LIN {X 0,Y 314.134,Z 385.842,A -85,B 0,C 180,E1 15646.01,E2 15646.01} C_VEL
LIN {X 0,Y 314.107,Z 385.802,A -85,B 0,C 180,E1 15641.542,E2 15641.542} C_VEL
LIN {X 0,Y 314.101,Z 385.806,A -85,B 0,C 180,E1 15637.158,E2 15637.158} C_VEL
LIN {X 0,Y 314.157,Z 386.054,A -85,B 0,C 180,E1 15633.754,E2 15633.754} C_VEL
LIN {X 0,Y 314.307,Z 386.869,A -85,B 0,C 180,E1 15633.361,E2 15633.361} C_VEL
LIN {X 0,Y 316.062,Z 390.166,A -85,B 0,C 180,E1 15632.503,E2 15632.503} C_VEL
LIN {X 0,Y 319.649,Z 392.888,A -85,B 0,C 180,E1 15631.061,E2 15631.061} C_VEL
LIN {X 0,Y 322.025,Z 396.633,A -85,B 0,C 180,E1 15629.967,E2 15629.967} C_VEL
LIN {X 0,Y 324.957,Z 398.845,A -85,B 0,C 180,E1 15628.68,E2 15628.68} C_VEL
LIN {X 0,Y 325.868,Z 399.667,A -85,B 0,C 180,E1 15628.262,E2 15628.262} C_VEL
LIN {X 0,Y 328.379,Z 403.252,A -85,B 0,C 180,E1 15626.985,E2 15626.985} C_VEL
LIN {X 0,Y 331.763,Z 405.775,A -85,B 0,C 180,E1 15625.29,E2 15625.29} C_VEL
LIN {X 0,Y 332.732,Z 406.589,A -85,B 0,C 180,E1 15624.775,E2 15624.775} C_VEL
LIN {X 0,Y 335.377,Z 410.277,A -85,B 0,C 180,E1 15623.197,E2 15623.197} C_VEL
LIN {X 0,Y 338.842,Z 412.794,A -85,B 0,C 180,E1 15621.168,E2 15621.168} C_VEL
LIN {X 0,Y 342.057,Z 417.138,A -85,B 0,C 180,E1 15619.111,E2 15619.111} C_VEL
LIN {X 0,Y 345.607,Z 419.696,A -85,B 0,C 180,E1 15616.954,E2 15616.954} C_VEL
LIN {X 0,Y 349.278,Z 424.393,A -85,B 0,C 180,E1 15614.534,E2 15614.534} C_VEL
LIN {X 0,Y 352.998,Z 427.12,A -85,B 0,C 180,E1 15612.104,E2 15612.104} C_VEL
LIN {X 0,Y 355.556,Z 430.698,A -85,B 0,C 180,E1 15610.256,E2 15610.256} C_VEL
LIN {X 0,Y 358.853,Z 433.234,A -85,B 0,C 180,E1 15607.97,E2 15607.97} C_VEL
LIN {X 0,Y 360.061,Z 434.113,A -85,B 0,C 180,E1 15607.103,E2 15607.103} C_VEL
LIN {X 0,Y 362.743,Z 437.733,A -85,B 0,C 180,E1 15604.981,E2 15604.981} C_VEL
LIN {X 0,Y 365.748,Z 440.111,A -85,B 0,C 180,E1 15602.668,E2 15602.668} C_VEL
LIN {X 0,Y 367.537,Z 441.34,A -85,B 0,C 180,E1 15601.213,E2 15601.213} C_VEL
LIN {X 0,Y 369.942,Z 444.728,A -85,B 0,C 180,E1 15599.021,E2 15599.021} C_VEL
LIN {X 0,Y 372.763,Z 447.045,A -85,B 0,C 180,E1 15596.401,E2 15596.401} C_VEL
LIN {X 0,Y 375.125,Z 448.378,A -85,B 0,C 180,E1 15594.15,E2 15594.15} C_VEL
LIN {X 0,Y 377.09,Z 451.528,A -85,B 0,C 180,E1 15591.79,E2 15591.79} C_VEL
LIN {X 0,Y 379.57,Z 453.798,A -85,B 0,C 180,E1 15588.745,E2 15588.745} C_VEL
LIN {X 0,Y 381.929,Z 454.969,A -85,B 0,C 180,E1 15585.487,E2 15585.487} C_VEL
LIN {X 0,Y 383.246,Z 456.112,A -85,B 0,C 180,E1 15583.272,E2 15583.272} C_VEL
LIN {X 0,Y 384.548,Z 458.408,A -85,B 0,C 180,E1 15580.335,E2 15580.335} C_VEL
LIN {X 0,Y 385.649,Z 459.744,A -85,B 0,C 180,E1 15577.149,E2 15577.149} C_VEL
LIN {X 0,Y 386.449,Z 460.442,A -85,B 0,C 180,E1 15573.709,E2 15573.709} C_VEL
LIN {X 0,Y 386.727,Z 460.669,A -85,B 0,C 180,E1 15570.444,E2 15570.444} C_VEL
LIN {X 0,Y 386.569,Z 460.508,A -85,B 0,C 180,E1 15567.035,E2 15567.035} C_VEL
LIN {X 0,Y 385.909,Z 459.957,A -85,B 0,C 180,E1 15563.604,E2 15563.604} C_VEL
LIN {X 0,Y 384.821,Z 458.695,A -85,B 0,C 180,E1 15560.277,E2 15560.277} C_VEL
LIN {X 0,Y 383.571,Z 456.693,A -85,B 0,C 180,E1 15557.352,E2 15557.352} C_VEL
LIN {X 0,Y 382.353,Z 455.172,A -85,B 0,C 180,E1 15555.152,E2 15555.152} C_VEL
LIN {X 0,Y 380.089,Z 454.101,A -85,B 0,C 180,E1 15551.917,E2 15551.917} C_VEL
LIN {X 0,Y 377.688,Z 452.178,A -85,B 0,C 180,E1 15548.898,E2 15548.898} C_VEL
LIN {X 0,Y 375.609,Z 449.353,A -85,B 0,C 180,E1 15546.467,E2 15546.467} C_VEL
LIN {X 0,Y 374.66,Z 447.969,A -85,B 0,C 180,E1 15545.398,E2 15545.398} C_VEL
LIN {X 0,Y 371.406,Z 446.102,A -85,B 0,C 180,E1 15542.315,E2 15542.315} C_VEL
LIN {X 0,Y 368.613,Z 443.116,A -85,B 0,C 180,E1 15539.791,E2 15539.791} C_VEL
LIN {X 0,Y 367.145,Z 440.822,A -85,B 0,C 180,E1 15538.454,E2 15538.454} C_VEL
LIN {X 0,Y 363.643,Z 438.62,A -85,B 0,C 180,E1 15535.692,E2 15535.692} C_VEL
LIN {X 0,Y 360.504,Z 434.893,A -85,B 0,C 180,E1 15533.26,E2 15533.26} C_VEL
LIN {X 0,Y 359.525,Z 433.574,A -85,B 0,C 180,E1 15532.48,E2 15532.48} C_VEL
LIN {X 0,Y 355.99,Z 431.139,A -85,B 0,C 180,E1 15530.048,E2 15530.048} C_VEL
LIN {X 0,Y 353.199,Z 427.491,A -85,B 0,C 180,E1 15528.048,E2 15528.048} C_VEL
LIN {X 0,Y 352.452,Z 426.566,A -85,B 0,C 180,E1 15527.511,E2 15527.511} C_VEL
LIN {X 0,Y 349.115,Z 424.229,A -85,B 0,C 180,E1 15525.359,E2 15525.359} C_VEL
LIN {X 0,Y 346.031,Z 420.14,A -85,B 0,C 180,E1 15523.309,E2 15523.309} C_VEL
LIN {X 0,Y 341.774,Z 416.854,A -85,B 0,C 180,E1 15520.708,E2 15520.708} C_VEL
LIN {X 0,Y 339.259,Z 413.179,A -85,B 0,C 180,E1 15519.089,E2 15519.089} C_VEL
LIN {X 0,Y 335.231,Z 410.123,A -85,B 0,C 180,E1 15516.715,E2 15516.715} C_VEL
LIN {X 0,Y 332.601,Z 406.366,A -85,B 0,C 180,E1 15515.149,E2 15515.149} C_VEL
LIN {X 0,Y 328.555,Z 403.427,A -85,B 0,C 180,E1 15513.099,E2 15513.099} C_VEL
LIN {X 0,Y 325.951,Z 399.829,A -85,B 0,C 180,E1 15511.781,E2 15511.781} C_VEL
LIN {X 0,Y 325.335,Z 399.029,A -85,B 0,C 180,E1 15511.486,E2 15511.486} C_VEL
LIN {X 0,Y 322.117,Z 396.737,A -85,B 0,C 180,E1 15510.075,E2 15510.075} C_VEL
LIN {X 0,Y 319.735,Z 393.08,A -85,B 0,C 180,E1 15508.982,E2 15508.982} C_VEL
LIN {X 0,Y 318.802,Z 392.189,A -85,B 0,C 180,E1 15508.581,E2 15508.581} C_VEL
LIN {X 0,Y 315.759,Z 389.81,A -85,B 0,C 180,E1 15507.372,E2 15507.372} C_VEL
LIN {X 0,Y 314.197,Z 386.347,A -85,B 0,C 180,E1 15506.446,E2 15506.446} C_VEL
LIN {X 0,Y 314.105,Z 385.806,A -85,B 0,C 180,E1 15505.238,E2 15505.238} C_VEL
LIN {X 0,Y 314.109,Z 385.86,A -85,B 0,C 180,E1 15500.639,E2 15500.639} C_VEL
LIN {X 0,Y 314.113,Z 385.793,A -85,B 0,C 180,E1 15496.258,E2 15496.258} C_VEL
LIN {X 0,Y 314.128,Z 385.82,A -85,B 0,C 180,E1 15491.931,E2 15491.931} C_VEL
LIN {X 0,Y 314.112,Z 385.804,A -85,B 0,C 180,E1 15491.223,E2 15491.223} C_VEL
LIN {X 0,Y 313.096,Z 385.927,A -85,B 0,C 180,E1 15489.818,E2 15489.818} C_VEL
LIN {X 0,Y 308.524,Z 386.553,A -85,B 0,C 180,E1 15487.159,E2 15487.159} C_VEL
LIN {X 0,Y 306.317,Z 386.828,A -85,B 0,C 180,E1 15485.321,E2 15485.321} C_VEL
LIN {X 0,Y 306.169,Z 386.831,A -85,B 0,C 180,E1 15484.797,E2 15484.797} C_VEL
LIN {X 0,Y 306.166,Z 386.781,A -85,B 0,C 180,E1 15480.179,E2 15480.179} C_VEL
LIN {X 0,Y 306.179,Z 386.801,A -85,B 0,C 180,E1 15475.872,E2 15475.872} C_VEL
LIN {X 0,Y 306.199,Z 386.796,A -85,B 0,C 180,E1 15471.353,E2 15471.353} C_VEL
LIN {X 0,Y 306.181,Z 386.781,A -85,B 0,C 180,E1 15466.971,E2 15466.971} C_VEL
LIN {X 0,Y 306.171,Z 386.841,A -85,B 0,C 180,E1 15462.509,E2 15462.509} C_VEL
LIN {X 0,Y 306.169,Z 386.801,A -85,B 0,C 180,E1 15457.934,E2 15457.934} C_VEL
LIN {X 0,Y 306.278,Z 387.264,A -85,B 0,C 180,E1 15457.133,E2 15457.133} C_VEL
LIN {X 0,Y 306.862,Z 389.204,A -85,B 0,C 180,E1 15456.519,E2 15456.519} C_VEL
LIN {X 0,Y 308.913,Z 391.919,A -85,B 0,C 180,E1 15455.518,E2 15455.518} C_VEL
LIN {X 0,Y 311.629,Z 393.769,A -85,B 0,C 180,E1 15454.357,E2 15454.357} C_VEL
LIN {X 0,Y 313.848,Z 397.415,A -85,B 0,C 180,E1 15453.352,E2 15453.352} C_VEL
LIN {X 0,Y 316.792,Z 399.976,A -85,B 0,C 180,E1 15452.197,E2 15452.197} C_VEL
LIN {X 0,Y 319.582,Z 404.027,A -85,B 0,C 180,E1 15451.087,E2 15451.087} C_VEL
LIN {X 0,Y 321.805,Z 406.272,A -85,B 0,C 180,E1 15450.286,E2 15450.286} C_VEL
LIN {X 0,Y 325.157,Z 410.566,A -85,B 0,C 180,E1 15449.095,E2 15449.095} C_VEL
LIN {X 0,Y 331.755,Z 420.166,A -85,B 0,C 180,E1 15446.883,E2 15446.883} C_VEL
LIN {X 0,Y 336.554,Z 427.526,A -85,B 0,C 180,E1 15445.39,E2 15445.39} C_VEL
LIN {X 0,Y 343.529,Z 438.829,A -85,B 0,C 180,E1 15443.363,E2 15443.363} C_VEL
LIN {X 0,Y 351.49,Z 452.715,A -85,B 0,C 180,E1 15441.22,E2 15441.22} C_VEL
LIN {X 0,Y 360.118,Z 469.418,A -85,B 0,C 180,E1 15439.056,E2 15439.056} C_VEL
LIN {X 0,Y 361.705,Z 473.056,A -85,B 0,C 180,E1 15438.662,E2 15438.662} C_VEL
LIN {X 0,Y 353.067,Z 645.3,A -85,B 0,C 180,E1 15435.126,E2 15435.126} C_VEL
LIN {X 0,Y 350.952,Z 666.531,A -85,B 0,C 180,E1 15434.485,E2 15434.485} C_VEL
LIN {X 0,Y 348.212,Z 685.14,A -85,B 0,C 180,E1 15433.674,E2 15433.674} C_VEL
LIN {X 0,Y 345.366,Z 701.117,A -85,B 0,C 180,E1 15432.779,E2 15432.779} C_VEL
LIN {X 0,Y 341.417,Z 720.205,A -85,B 0,C 180,E1 15431.44,E2 15431.44} C_VEL
LIN {X 0,Y 337.052,Z 737.957,A -85,B 0,C 180,E1 15429.847,E2 15429.847} C_VEL
LIN {X 0,Y 332.99,Z 753.101,A -85,B 0,C 180,E1 15428.209,E2 15428.209} C_VEL
LIN {X 0,Y 328.131,Z 769.951,A -85,B 0,C 180,E1 15426.021,E2 15426.021} C_VEL
LIN {X 0,Y 323.55,Z 784.594,A -85,B 0,C 180,E1 15423.689,E2 15423.689} C_VEL
LIN {X 0,Y 319.787,Z 796.417,A -85,B 0,C 180,E1 15421.475,E2 15421.475} C_VEL
LIN {X 0,Y 315.618,Z 809.568,A -85,B 0,C 180,E1 15418.577,E2 15418.577} C_VEL
LIN {X 0,Y 311.951,Z 821.161,A -85,B 0,C 180,E1 15415.435,E2 15415.435} C_VEL
LIN {X 0,Y 309.368,Z 829.915,A -85,B 0,C 180,E1 15412.618,E2 15412.618} C_VEL
LIN {X 0,Y 307.027,Z 838.857,A -85,B 0,C 180,E1 15409.181,E2 15409.181} C_VEL
LIN {X 0,Y 305.383,Z 846.223,A -85,B 0,C 180,E1 15405.573,E2 15405.573} C_VEL
LIN {X 0,Y 304.505,Z 851.46,A -85,B 0,C 180,E1 15402.323,E2 15402.323} C_VEL
LIN {X 0,Y 304.088,Z 855.451,A -85,B 0,C 180,E1 15399.081,E2 15399.081} C_VEL
LIN {X 0,Y 303.953,Z 858.609,A -85,B 0,C 180,E1 15395.285,E2 15395.285} C_VEL
LIN {X 0,Y 303.966,Z 859.939,A -85,B 0,C 180,E1 15391.885,E2 15391.885} C_VEL
LIN {X 0,Y 303.973,Z 860.058,A -85,B 0,C 180,E1 15388.869,E2 15388.869} C_VEL
LIN {X 0,Y 303.951,Z 859.146,A -85,B 0,C 180,E1 15385.85,E2 15385.85} C_VEL
LIN {X 0,Y 303.996,Z 857.197,A -85,B 0,C 180,E1 15382.82,E2 15382.82} C_VEL
LIN {X 0,Y 304.26,Z 853.559,A -85,B 0,C 180,E1 15379.204,E2 15379.204} C_VEL
LIN {X 0,Y 305.068,Z 847.903,A -85,B 0,C 180,E1 15375.383,E2 15375.383} C_VEL
LIN {X 0,Y 306.241,Z 842.09,A -85,B 0,C 180,E1 15372.324,E2 15372.324} C_VEL
LIN {X 0,Y 308.009,Z 834.909,A -85,B 0,C 180,E1 15369.225,E2 15369.225} C_VEL
LIN {X 0,Y 311.058,Z 824.166,A -85,B 0,C 180,E1 15365.47,E2 15365.47} C_VEL
LIN {X 0,Y 314.227,Z 813.813,A -85,B 0,C 180,E1 15362.524,E2 15362.524} C_VEL
LIN {X 0,Y 317.873,Z 802.427,A -85,B 0,C 180,E1 15359.784,E2 15359.784} C_VEL
LIN {X 0,Y 322.462,Z 788.102,A -85,B 0,C 180,E1 15356.927,E2 15356.927} C_VEL
LIN {X 0,Y 326.535,Z 775.009,A -85,B 0,C 180,E1 15354.748,E2 15354.748} C_VEL
LIN {X 0,Y 330.675,Z 761.195,A -85,B 0,C 180,E1 15352.791,E2 15352.791} C_VEL
LIN {X 0,Y 335.814,Z 742.802,A -85,B 0,C 180,E1 15350.641,E2 15350.641} C_VEL
LIN {X 0,Y 339.765,Z 727.054,A -85,B 0,C 180,E1 15349.145,E2 15349.145} C_VEL
LIN {X 0,Y 343.217,Z 711.73,A -85,B 0,C 180,E1 15347.932,E2 15347.932} C_VEL
LIN {X 0,Y 347.068,Z 692.121,A -85,B 0,C 180,E1 15346.68,E2 15346.68} C_VEL
LIN {X 0,Y 350.049,Z 672.91,A -85,B 0,C 180,E1 15345.769,E2 15345.769} C_VEL
LIN {X 0,Y 352.175,Z 655.468,A -85,B 0,C 180,E1 15345.153,E2 15345.153} C_VEL
LIN {X 0,Y 353.864,Z 632.381,A -85,B 0,C 180,E1 15344.579,E2 15344.579} C_VEL
LIN {X 0,Y 361.643,Z 472.564,A -85,B 0,C 180,E1 15341.312,E2 15341.312} C_VEL
LIN {X 0,Y 353.02,Z 455.542,A -85,B 0,C 180,E1 15339.174,E2 15339.174} C_VEL
LIN {X 0,Y 344.501,Z 440.417,A -85,B 0,C 180,E1 15336.906,E2 15336.906} C_VEL
LIN {X 0,Y 337.468,Z 428.931,A -85,B 0,C 180,E1 15334.884,E2 15334.884} C_VEL
LIN {X 0,Y 332.59,Z 421.431,A -85,B 0,C 180,E1 15333.383,E2 15333.383} C_VEL
LIN {X 0,Y 325.496,Z 410.902,A -85,B 0,C 180,E1 15331.018,E2 15331.018} C_VEL
LIN {X 0,Y 321.91,Z 406.453,A -85,B 0,C 180,E1 15329.755,E2 15329.755} C_VEL
LIN {X 0,Y 320.697,Z 405.041,A -85,B 0,C 180,E1 15329.314,E2 15329.314} C_VEL
LIN {X 0,Y 317.579,Z 401.425,A -85,B 0,C 180,E1 15328.136,E2 15328.136} C_VEL
LIN {X 0,Y 316.267,Z 399.428,A -85,B 0,C 180,E1 15327.597,E2 15327.597} C_VEL
LIN {X 0,Y 313.156,Z 396.551,A -85,B 0,C 180,E1 15326.354,E2 15326.354} C_VEL
LIN {X 0,Y 311.307,Z 393.355,A -85,B 0,C 180,E1 15325.499,E2 15325.499} C_VEL
LIN {X 0,Y 308.073,Z 391.089,A -85,B 0,C 180,E1 15324.094,E2 15324.094} C_VEL
LIN {X 0,Y 306.327,Z 387.548,A -85,B 0,C 180,E1 15323.011,E2 15323.011} C_VEL
LIN {X 0,Y 306.177,Z 386.826,A -85,B 0,C 180,E1 15322.267,E2 15322.267} C_VEL
LIN {X 0,Y 306.169,Z 386.847,A -85,B 0,C 180,E1 15317.688,E2 15317.688} C_VEL
LIN {X 0,Y 306.173,Z 386.78,A -85,B 0,C 180,E1 15313.222,E2 15313.222} C_VEL
LIN {X 0,Y 306.191,Z 386.802,A -85,B 0,C 180,E1 15308.836,E2 15308.836} C_VEL
LIN {X 0,Y 306.191,Z 386.79,A -85,B 0,C 180,E1 15304.503,E2 15304.503} C_VEL
LIN {X 0,Y 306.186,Z 386.786,A -85,B 0,C 180,E1 15300.195,E2 15300.195} C_VEL
LIN {X 0,Y 306.169,Z 386.813,A -85,B 0,C 180,E1 15295.701,E2 15295.701} C_VEL
LIN {X 0,Y 306.161,Z 386.776,A -85,B 0,C 180,E1 15291.18,E2 15291.18} C_VEL
LIN {X 0,Y 306.187,Z 386.847,A -85,B 0,C 180,E1 15286.603,E2 15286.603} C_VEL
LIN {X 0,Y 306.194,Z 386.779,A -85,B 0,C 180,E1 15282.134,E2 15282.134} C_VEL
LIN {X 0,Y 306.183,Z 386.801,A -85,B 0,C 180,E1 15277.751,E2 15277.751} C_VEL
LIN {X 0,Y 306.241,Z 387.267,A -85,B 0,C 180,E1 15276.741,E2 15276.741} C_VEL
LIN {X 0,Y 306.751,Z 388.881,A -85,B 0,C 180,E1 15276.171,E2 15276.171} C_VEL
LIN {X 0,Y 308.679,Z 391.684,A -85,B 0,C 180,E1 15275.21,E2 15275.21} C_VEL
LIN {X 0,Y 311.576,Z 393.761,A -85,B 0,C 180,E1 15273.962,E2 15273.962} C_VEL
LIN {X 0,Y 313.793,Z 397.424,A -85,B 0,C 180,E1 15272.956,E2 15272.956} C_VEL
LIN {X 0,Y 317.418,Z 400.388,A -85,B 0,C 180,E1 15271.507,E2 15271.507} C_VEL
LIN {X 0,Y 320.252,Z 404.323,A -85,B 0,C 180,E1 15270.248,E2 15270.248} C_VEL
LIN {X 0,Y 323.778,Z 407.065,A -85,B 0,C 180,E1 15268.708,E2 15268.708} C_VEL
LIN {X 0,Y 326.587,Z 410.821,A -85,B 0,C 180,E1 15267.314,E2 15267.314} C_VEL
LIN {X 0,Y 329.898,Z 413.342,A -85,B 0,C 180,E1 15265.698,E2 15265.698} C_VEL
LIN {X 0,Y 331.04,Z 414.305,A -85,B 0,C 180,E1 15265.097,E2 15265.097} C_VEL
LIN {X 0,Y 333.916,Z 418.027,A -85,B 0,C 180,E1 15263.437,E2 15263.437} C_VEL
LIN {X 0,Y 337.812,Z 421.112,A -85,B 0,C 180,E1 15261.148,E2 15261.148} C_VEL
LIN {X 0,Y 340.503,Z 424.745,A -85,B 0,C 180,E1 15259.44,E2 15259.44} C_VEL
LIN {X 0,Y 344.613,Z 428.027,A -85,B 0,C 180,E1 15256.914,E2 15256.914} C_VEL
LIN {X 0,Y 347.882,Z 432.151,A -85,B 0,C 180,E1 15254.76,E2 15254.76} C_VEL
LIN {X 0,Y 351.622,Z 434.96,A -85,B 0,C 180,E1 15252.341,E2 15252.341} C_VEL
LIN {X 0,Y 354.583,Z 438.839,A -85,B 0,C 180,E1 15250.22,E2 15250.22} C_VEL
LIN {X 0,Y 358.084,Z 441.324,A -85,B 0,C 180,E1 15247.812,E2 15247.812} C_VEL
LIN {X 0,Y 359.032,Z 442.437,A -85,B 0,C 180,E1 15247.09,E2 15247.09} C_VEL
LIN {X 0,Y 362.151,Z 446.226,A -85,B 0,C 180,E1 15244.658,E2 15244.658} C_VEL
LIN {X 0,Y 365.541,Z 448.482,A -85,B 0,C 180,E1 15242.031,E2 15242.031} C_VEL
LIN {X 0,Y 366.425,Z 449.431,A -85,B 0,C 180,E1 15241.282,E2 15241.282} C_VEL
LIN {X 0,Y 369.01,Z 452.821,A -85,B 0,C 180,E1 15238.954,E2 15238.954} C_VEL
LIN {X 0,Y 371.841,Z 455.035,A -85,B 0,C 180,E1 15236.338,E2 15236.338} C_VEL
LIN {X 0,Y 373.984,Z 456.292,A -85,B 0,C 180,E1 15234.288,E2 15234.288} C_VEL
LIN {X 0,Y 376.044,Z 459.474,A -85,B 0,C 180,E1 15231.853,E2 15231.853} C_VEL
LIN {X 0,Y 378.549,Z 461.727,A -85,B 0,C 180,E1 15228.798,E2 15228.798} C_VEL
LIN {X 0,Y 380.923,Z 462.9,A -85,B 0,C 180,E1 15225.529,E2 15225.529} C_VEL
LIN {X 0,Y 382.213,Z 464.043,A -85,B 0,C 180,E1 15223.355,E2 15223.355} C_VEL
LIN {X 0,Y 383.559,Z 466.349,A -85,B 0,C 180,E1 15220.362,E2 15220.362} C_VEL
LIN {X 0,Y 384.666,Z 467.687,A -85,B 0,C 180,E1 15217.167,E2 15217.167} C_VEL
LIN {X 0,Y 385.473,Z 468.382,A -85,B 0,C 180,E1 15213.718,E2 15213.718} C_VEL
LIN {X 0,Y 385.752,Z 468.61,A -85,B 0,C 180,E1 15210.446,E2 15210.446} C_VEL
LIN {X 0,Y 385.591,Z 468.448,A -85,B 0,C 180,E1 15207.027,E2 15207.027} C_VEL
LIN {X 0,Y 384.927,Z 467.896,A -85,B 0,C 180,E1 15203.587,E2 15203.587} C_VEL
LIN {X 0,Y 383.832,Z 466.645,A -85,B 0,C 180,E1 15200.252,E2 15200.252} C_VEL
LIN {X 0,Y 382.575,Z 464.657,A -85,B 0,C 180,E1 15197.319,E2 15197.319} C_VEL
LIN {X 0,Y 381.344,Z 463.104,A -85,B 0,C 180,E1 15195.111,E2 15195.111} C_VEL
LIN {X 0,Y 378.962,Z 461.981,A -85,B 0,C 180,E1 15191.74,E2 15191.74} C_VEL
LIN {X 0,Y 376.492,Z 459.963,A -85,B 0,C 180,E1 15188.665,E2 15188.665} C_VEL
LIN {X 0,Y 374.332,Z 456.954,A -85,B 0,C 180,E1 15186.131,E2 15186.131} C_VEL
LIN {X 0,Y 373.588,Z 455.884,A -85,B 0,C 180,E1 15185.323,E2 15185.323} C_VEL
LIN {X 0,Y 370.207,Z 453.938,A -85,B 0,C 180,E1 15182.146,E2 15182.146} C_VEL
LIN {X 0,Y 367.386,Z 450.924,A -85,B 0,C 180,E1 15179.589,E2 15179.589} C_VEL
LIN {X 0,Y 365.776,Z 448.603,A -85,B 0,C 180,E1 15178.16,E2 15178.16} C_VEL
LIN {X 0,Y 362.296,Z 446.36,A -85,B 0,C 180,E1 15175.448,E2 15175.448} C_VEL
LIN {X 0,Y 359.161,Z 442.65,A -85,B 0,C 180,E1 15173.015,E2 15173.015} C_VEL
LIN {X 0,Y 358.305,Z 441.431,A -85,B 0,C 180,E1 15172.331,E2 15172.331} C_VEL
LIN {X 0,Y 354.623,Z 438.881,A -85,B 0,C 180,E1 15169.81,E2 15169.81} C_VEL
LIN {X 0,Y 351.686,Z 435.077,A -85,B 0,C 180,E1 15167.708,E2 15167.708} C_VEL
LIN {X 0,Y 350.719,Z 434.178,A -85,B 0,C 180,E1 15167.052,E2 15167.052} C_VEL
LIN {X 0,Y 347.384,Z 431.656,A -85,B 0,C 180,E1 15164.925,E2 15164.925} C_VEL
LIN {X 0,Y 343.932,Z 427.341,A -85,B 0,C 180,E1 15162.652,E2 15162.652} C_VEL
LIN {X 0,Y 340.084,Z 424.302,A -85,B 0,C 180,E1 15160.288,E2 15160.288} C_VEL
LIN {X 0,Y 337.251,Z 420.482,A -85,B 0,C 180,E1 15158.493,E2 15158.493} C_VEL
LIN {X 0,Y 333.606,Z 417.721,A -85,B 0,C 180,E1 15156.389,E2 15156.389} C_VEL
LIN {X 0,Y 330.582,Z 413.692,A -85,B 0,C 180,E1 15154.642,E2 15154.642} C_VEL
LIN {X 0,Y 326.953,Z 411.18,A -85,B 0,C 180,E1 15152.864,E2 15152.864} C_VEL
LIN {X 0,Y 324.029,Z 407.5,A -85,B 0,C 180,E1 15151.42,E2 15151.42} C_VEL
LIN {X 0,Y 323.239,Z 406.522,A -85,B 0,C 180,E1 15151.041,E2 15151.041} C_VEL
LIN {X 0,Y 319.862,Z 403.917,A -85,B 0,C 180,E1 15149.585,E2 15149.585} C_VEL
LIN {X 0,Y 316.805,Z 399.756,A -85,B 0,C 180,E1 15148.245,E2 15148.245} C_VEL
LIN {X 0,Y 313.394,Z 396.952,A -85,B 0,C 180,E1 15146.877,E2 15146.877} C_VEL
LIN {X 0,Y 311.254,Z 393.35,A -85,B 0,C 180,E1 15145.894,E2 15145.894} C_VEL
LIN {X 0,Y 308.031,Z 391,A -85,B 0,C 180,E1 15144.488,E2 15144.488} C_VEL
LIN {X 0,Y 306.326,Z 387.628,A -85,B 0,C 180,E1 15143.456,E2 15143.456} C_VEL
LIN {X 0,Y 306.172,Z 386.852,A -85,B 0,C 180,E1 15142.655,E2 15142.655} C_VEL
LIN {X 0,Y 306.183,Z 386.783,A -85,B 0,C 180,E1 15138.149,E2 15138.149} C_VEL
LIN {X 0,Y 306.198,Z 386.842,A -85,B 0,C 180,E1 15133.589,E2 15133.589} C_VEL
LIN {X 0,Y 306.165,Z 386.774,A -85,B 0,C 180,E1 15129.01,E2 15129.01} C_VEL
LIN {X 0,Y 306.169,Z 386.831,A -85,B 0,C 180,E1 15124.797,E2 15124.797} C_VEL
LIN {X 0,Y 305.16,Z 386.914,A -85,B 0,C 180,E1 15123.355,E2 15123.355} C_VEL
LIN {X 0,Y 300.723,Z 387.451,A -85,B 0,C 180,E1 15120.729,E2 15120.729} C_VEL
LIN {X 0,Y 298.418,Z 387.775,A -85,B 0,C 180,E1 15118.846,E2 15118.846} C_VEL
LIN {X 0,Y 298.234,Z 387.82,A -85,B 0,C 180,E1 15118.2,E2 15118.2} C_VEL
LIN {X 0,Y 298.251,Z 387.756,A -85,B 0,C 180,E1 15113.64,E2 15113.64} C_VEL
LIN {X 0,Y 298.254,Z 387.821,A -85,B 0,C 180,E1 15109.172,E2 15109.172} C_VEL
LIN {X 0,Y 298.23,Z 387.771,A -85,B 0,C 180,E1 15104.634,E2 15104.634} C_VEL
LIN {X 0,Y 298.285,Z 387.974,A -85,B 0,C 180,E1 15101.221,E2 15101.221} C_VEL
LIN {X 0,Y 298.564,Z 389.281,A -85,B 0,C 180,E1 15100.478,E2 15100.478} C_VEL
LIN {X 0,Y 300.194,Z 392.079,A -85,B 0,C 180,E1 15099.42,E2 15099.42} C_VEL
LIN {X 0,Y 303.438,Z 394.346,A -85,B 0,C 180,E1 15097.725,E2 15097.725} C_VEL
LIN {X 0,Y 304.184,Z 395.41,A -85,B 0,C 180,E1 15097.324,E2 15097.324} C_VEL
LIN {X 0,Y 306.293,Z 398.749,A -85,B 0,C 180,E1 15096.218,E2 15096.218} C_VEL
LIN {X 0,Y 309.355,Z 401.238,A -85,B 0,C 180,E1 15094.841,E2 15094.841} C_VEL
LIN {X 0,Y 312.091,Z 405.212,A -85,B 0,C 180,E1 15093.601,E2 15093.601} C_VEL
LIN {X 0,Y 314.461,Z 407.476,A -85,B 0,C 180,E1 15092.642,E2 15092.642} C_VEL
LIN {X 0,Y 317.664,Z 411.714,A -85,B 0,C 180,E1 15091.359,E2 15091.359} C_VEL
LIN {X 0,Y 319.294,Z 413.543,A -85,B 0,C 180,E1 15090.751,E2 15090.751} C_VEL
LIN {X 0,Y 324.393,Z 420.293,A -85,B 0,C 180,E1 15088.911,E2 15088.911} C_VEL
LIN {X 0,Y 332.54,Z 432.789,A -85,B 0,C 180,E1 15086.197,E2 15086.197} C_VEL
LIN {X 0,Y 339.939,Z 445.035,A -85,B 0,C 180,E1 15083.96,E2 15083.96} C_VEL
LIN {X 0,Y 347.616,Z 458.718,A -85,B 0,C 180,E1 15081.82,E2 15081.82} C_VEL
LIN {X 0,Y 355.977,Z 475.255,A -85,B 0,C 180,E1 15079.647,E2 15079.647} C_VEL
LIN {X 0,Y 356.256,Z 476.515,A -85,B 0,C 180,E1 15079.556,E2 15079.556} C_VEL
LIN {X 0,Y 347.447,Z 645.097,A -85,B 0,C 180,E1 15076.063,E2 15076.063} C_VEL
LIN {X 0,Y 345.264,Z 666.317,A -85,B 0,C 180,E1 15075.418,E2 15075.418} C_VEL
LIN {X 0,Y 342.437,Z 684.902,A -85,B 0,C 180,E1 15074.604,E2 15074.604} C_VEL
LIN {X 0,Y 339.529,Z 700.681,A -85,B 0,C 180,E1 15073.716,E2 15073.716} C_VEL
LIN {X 0,Y 335.627,Z 718.938,A -85,B 0,C 180,E1 15072.434,E2 15072.434} C_VEL
LIN {X 0,Y 331.081,Z 736.91,A -85,B 0,C 180,E1 15070.829,E2 15070.829} C_VEL
LIN {X 0,Y 327.04,Z 751.435,A -85,B 0,C 180,E1 15069.26,E2 15069.26} C_VEL
LIN {X 0,Y 322.484,Z 766.64,A -85,B 0,C 180,E1 15067.31,E2 15067.31} C_VEL
LIN {X 0,Y 317.11,Z 783.351,A -85,B 0,C 180,E1 15064.688,E2 15064.688} C_VEL
LIN {X 0,Y 312.817,Z 796.174,A -85,B 0,C 180,E1 15062.26,E2 15062.26} C_VEL
LIN {X 0,Y 308.397,Z 809.419,A -85,B 0,C 180,E1 15059.284,E2 15059.284} C_VEL
LIN {X 0,Y 304.549,Z 820.918,A -85,B 0,C 180,E1 15056.099,E2 15056.099} C_VEL
LIN {X 0,Y 301.8,Z 829.672,A -85,B 0,C 180,E1 15053.218,E2 15053.218} C_VEL
LIN {X 0,Y 299.307,Z 838.564,A -85,B 0,C 180,E1 15049.718,E2 15049.718} C_VEL
LIN {X 0,Y 297.523,Z 845.982,A -85,B 0,C 180,E1 15045.995,E2 15045.995} C_VEL
LIN {X 0,Y 296.569,Z 851.22,A -85,B 0,C 180,E1 15042.658,E2 15042.658} C_VEL
LIN {X 0,Y 296.107,Z 855.212,A -85,B 0,C 180,E1 15039.327,E2 15039.327} C_VEL
LIN {X 0,Y 295.956,Z 858.372,A -85,B 0,C 180,E1 15035.428,E2 15035.428} C_VEL
LIN {X 0,Y 295.968,Z 859.702,A -85,B 0,C 180,E1 15031.936,E2 15031.936} C_VEL
LIN {X 0,Y 295.977,Z 859.821,A -85,B 0,C 180,E1 15028.839,E2 15028.839} C_VEL
LIN {X 0,Y 295.952,Z 858.909,A -85,B 0,C 180,E1 15025.738,E2 15025.738} C_VEL
LIN {X 0,Y 296.002,Z 856.959,A -85,B 0,C 180,E1 15022.625,E2 15022.625} C_VEL
LIN {X 0,Y 296.298,Z 853.32,A -85,B 0,C 180,E1 15018.911,E2 15018.911} C_VEL
LIN {X 0,Y 297.198,Z 847.573,A -85,B 0,C 180,E1 15014.934,E2 15014.934} C_VEL
LIN {X 0,Y 298.548,Z 841.446,A -85,B 0,C 180,E1 15011.651,E2 15011.651} C_VEL
LIN {X 0,Y 300.808,Z 833.142,A -85,B 0,C 180,E1 15008.041,E2 15008.041} C_VEL
LIN {X 0,Y 303.949,Z 822.782,A -85,B 0,C 180,E1 15004.474,E2 15004.474} C_VEL
LIN {X 0,Y 307.194,Z 812.865,A -85,B 0,C 180,E1 15001.628,E2 15001.628} C_VEL
LIN {X 0,Y 311.378,Z 800.595,A -85,B 0,C 180,E1 14998.656,E2 14998.656} C_VEL
LIN {X 0,Y 316.107,Z 786.356,A -85,B 0,C 180,E1 14995.846,E2 14995.846} C_VEL
LIN {X 0,Y 320.258,Z 773.644,A -85,B 0,C 180,E1 14993.729,E2 14993.729} C_VEL
LIN {X 0,Y 325.231,Z 757.795,A -85,B 0,C 180,E1 14991.499,E2 14991.499} C_VEL
LIN {X 0,Y 329.994,Z 740.947,A -85,B 0,C 180,E1 14989.58,E2 14989.58} C_VEL
LIN {X 0,Y 333.997,Z 725.51,A -85,B 0,C 180,E1 14988.121,E2 14988.121} C_VEL
LIN {X 0,Y 338.23,Z 707.237,A -85,B 0,C 180,E1 14986.701,E2 14986.701} C_VEL
LIN {X 0,Y 341.951,Z 687.728,A -85,B 0,C 180,E1 14985.539,E2 14985.539} C_VEL
LIN {X 0,Y 344.603,Z 670.842,A -85,B 0,C 180,E1 14984.763,E2 14984.763} C_VEL
LIN {X 0,Y 347.043,Z 650.631,A -85,B 0,C 180,E1 14984.074,E2 14984.074} C_VEL
LIN {X 0,Y 349.015,Z 617.36,A -85,B 0,C 180,E1 14983.334,E2 14983.334} C_VEL
LIN {X 0,Y 356.18,Z 475.69,A -85,B 0,C 180,E1 14980.405,E2 14980.405} C_VEL
LIN {X 0,Y 347.943,Z 459.35,A -85,B 0,C 180,E1 14978.268,E2 14978.268} C_VEL
LIN {X 0,Y 340.319,Z 445.674,A -85,B 0,C 180,E1 14976.149,E2 14976.149} C_VEL
LIN {X 0,Y 333.623,Z 434.569,A -85,B 0,C 180,E1 14974.144,E2 14974.144} C_VEL
LIN {X 0,Y 328.868,Z 427.127,A -85,B 0,C 180,E1 14972.62,E2 14972.62} C_VEL
LIN {X 0,Y 322.491,Z 417.596,A -85,B 0,C 180,E1 14970.414,E2 14970.414} C_VEL
LIN {X 0,Y 318.215,Z 412.215,A -85,B 0,C 180,E1 14968.843,E2 14968.843} C_VEL
LIN {X 0,Y 314.851,Z 408.154,A -85,B 0,C 180,E1 14967.527,E2 14967.527} C_VEL
LIN {X 0,Y 313.642,Z 406.552,A -85,B 0,C 180,E1 14967.025,E2 14967.025} C_VEL
LIN {X 0,Y 310.44,Z 403.152,A -85,B 0,C 180,E1 14965.677,E2 14965.677} C_VEL
LIN {X 0,Y 308.98,Z 400.765,A -85,B 0,C 180,E1 14964.987,E2 14964.987} C_VEL
LIN {X 0,Y 305.756,Z 398.127,A -85,B 0,C 180,E1 14963.52,E2 14963.52} C_VEL
LIN {X 0,Y 303.62,Z 394.423,A -85,B 0,C 180,E1 14962.363,E2 14962.363} C_VEL
LIN {X 0,Y 300.353,Z 392.246,A -85,B 0,C 180,E1 14960.67,E2 14960.67} C_VEL
LIN {X 0,Y 298.62,Z 389.448,A -85,B 0,C 180,E1 14959.569,E2 14959.569} C_VEL
LIN {X 0,Y 298.311,Z 388.178,A -85,B 0,C 180,E1 14958.98,E2 14958.98} C_VEL
LIN {X 0,Y 298.252,Z 387.805,A -85,B 0,C 180,E1 14956.965,E2 14956.965} C_VEL
LIN {X 0,Y 298.255,Z 387.773,A -85,B 0,C 180,E1 14952.594,E2 14952.594} C_VEL
LIN {X 0,Y 298.235,Z 387.774,A -85,B 0,C 180,E1 14948.102,E2 14948.102} C_VEL
LIN {X 0,Y 298.226,Z 387.802,A -85,B 0,C 180,E1 14943.66,E2 14943.66} C_VEL
LIN {X 0,Y 298.227,Z 387.759,A -85,B 0,C 180,E1 14939.048,E2 14939.048} C_VEL
LIN {X 0,Y 298.262,Z 387.833,A -85,B 0,C 180,E1 14934.43,E2 14934.43} C_VEL
LIN {X 0,Y 298.24,Z 387.76,A -85,B 0,C 180,E1 14929.969,E2 14929.969} C_VEL
LIN {X 0,Y 298.227,Z 387.8,A -85,B 0,C 180,E1 14925.446,E2 14925.446} C_VEL
LIN {X 0,Y 298.246,Z 387.928,A -85,B 0,C 180,E1 14920.894,E2 14920.894} C_VEL
LIN {X 0,Y 298.572,Z 389.241,A -85,B 0,C 180,E1 14920.063,E2 14920.063} C_VEL
LIN {X 0,Y 300.147,Z 392.107,A -85,B 0,C 180,E1 14919.027,E2 14919.027} C_VEL
LIN {X 0,Y 303.999,Z 394.921,A -85,B 0,C 180,E1 14917.021,E2 14917.021} C_VEL
LIN {X 0,Y 306.164,Z 398.572,A -85,B 0,C 180,E1 14915.866,E2 14915.866} C_VEL
LIN {X 0,Y 309.307,Z 401.224,A -85,B 0,C 180,E1 14914.445,E2 14914.445} C_VEL
LIN {X 0,Y 311.941,Z 405.104,A -85,B 0,C 180,E1 14913.245,E2 14913.245} C_VEL
LIN {X 0,Y 315.24,Z 407.939,A -85,B 0,C 180,E1 14911.912,E2 14911.912} C_VEL
LIN {X 0,Y 318.345,Z 411.896,A -85,B 0,C 180,E1 14910.57,E2 14910.57} C_VEL
LIN {X 0,Y 321.935,Z 414.834,A -85,B 0,C 180,E1 14909.029,E2 14909.029} C_VEL
LIN {X 0,Y 325.185,Z 418.764,A -85,B 0,C 180,E1 14907.459,E2 14907.459} C_VEL
LIN {X 0,Y 329.266,Z 421.867,A -85,B 0,C 180,E1 14905.464,E2 14905.464} C_VEL
LIN {X 0,Y 332.429,Z 425.773,A -85,B 0,C 180,E1 14903.676,E2 14903.676} C_VEL
LIN {X 0,Y 336.237,Z 428.774,A -85,B 0,C 180,E1 14901.478,E2 14901.478} C_VEL
LIN {X 0,Y 339.233,Z 432.632,A -85,B 0,C 180,E1 14899.59,E2 14899.59} C_VEL
LIN {X 0,Y 343.124,Z 435.759,A -85,B 0,C 180,E1 14897.194,E2 14897.194} C_VEL
LIN {X 0,Y 346.477,Z 439.903,A -85,B 0,C 180,E1 14894.991,E2 14894.991} C_VEL
LIN {X 0,Y 350.185,Z 442.672,A -85,B 0,C 180,E1 14892.629,E2 14892.629} C_VEL
LIN {X 0,Y 353.315,Z 446.674,A -85,B 0,C 180,E1 14890.394,E2 14890.394} C_VEL
LIN {X 0,Y 356.712,Z 449.109,A -85,B 0,C 180,E1 14888.051,E2 14888.051} C_VEL
LIN {X 0,Y 357.823,Z 450.399,A -85,B 0,C 180,E1 14887.232,E2 14887.232} C_VEL
LIN {X 0,Y 361.09,Z 454.224,A -85,B 0,C 180,E1 14884.693,E2 14884.693} C_VEL
LIN {X 0,Y 365.031,Z 457.034,A -85,B 0,C 180,E1 14881.605,E2 14881.605} C_VEL
LIN {X 0,Y 367.714,Z 460.541,A -85,B 0,C 180,E1 14879.231,E2 14879.231} C_VEL
LIN {X 0,Y 370.714,Z 462.922,A -85,B 0,C 180,E1 14876.458,E2 14876.458} C_VEL
LIN {X 0,Y 372.785,Z 464.117,A -85,B 0,C 180,E1 14874.48,E2 14874.48} C_VEL
LIN {X 0,Y 374.858,Z 467.248,A -85,B 0,C 180,E1 14872.091,E2 14872.091} C_VEL
LIN {X 0,Y 377.408,Z 469.566,A -85,B 0,C 180,E1 14869.017,E2 14869.017} C_VEL
LIN {X 0,Y 379.892,Z 470.82,A -85,B 0,C 180,E1 14865.611,E2 14865.611} C_VEL
LIN {X 0,Y 381.148,Z 471.912,A -85,B 0,C 180,E1 14863.501,E2 14863.501} C_VEL
LIN {X 0,Y 382.57,Z 474.291,A -85,B 0,C 180,E1 14860.389,E2 14860.389} C_VEL
LIN {X 0,Y 383.684,Z 475.63,A -85,B 0,C 180,E1 14857.185,E2 14857.185} C_VEL
LIN {X 0,Y 384.496,Z 476.323,A -85,B 0,C 180,E1 14853.727,E2 14853.727} C_VEL
LIN {X 0,Y 384.777,Z 476.551,A -85,B 0,C 180,E1 14850.447,E2 14850.447} C_VEL
LIN {X 0,Y 384.613,Z 476.388,A -85,B 0,C 180,E1 14847.02,E2 14847.02} C_VEL
LIN {X 0,Y 383.985,Z 475.864,A -85,B 0,C 180,E1 14843.722,E2 14843.722} C_VEL
LIN {X 0,Y 382.891,Z 474.683,A -85,B 0,C 180,E1 14840.38,E2 14840.38} C_VEL
LIN {X 0,Y 381.639,Z 472.749,A -85,B 0,C 180,E1 14837.441,E2 14837.441} C_VEL
LIN {X 0,Y 380.335,Z 471.036,A -85,B 0,C 180,E1 14835.071,E2 14835.071} C_VEL
LIN {X 0,Y 377.96,Z 469.919,A -85,B 0,C 180,E1 14831.717,E2 14831.717} C_VEL
LIN {X 0,Y 375.444,Z 467.9,A -85,B 0,C 180,E1 14828.602,E2 14828.602} C_VEL
LIN {X 0,Y 373.199,Z 464.835,A -85,B 0,C 180,E1 14825.97,E2 14825.97} C_VEL
LIN {X 0,Y 372.321,Z 463.724,A -85,B 0,C 180,E1 14825.064,E2 14825.064} C_VEL
LIN {X 0,Y 369.052,Z 461.806,A -85,B 0,C 180,E1 14822.011,E2 14822.011} C_VEL
LIN {X 0,Y 366.096,Z 458.644,A -85,B 0,C 180,E1 14819.331,E2 14819.331} C_VEL
LIN {X 0,Y 364.503,Z 456.419,A -85,B 0,C 180,E1 14817.933,E2 14817.933} C_VEL
LIN {X 0,Y 360.961,Z 454.105,A -85,B 0,C 180,E1 14815.208,E2 14815.208} C_VEL
LIN {X 0,Y 357.689,Z 450.191,A -85,B 0,C 180,E1 14812.658,E2 14812.658} C_VEL
LIN {X 0,Y 356.677,Z 449.092,A -85,B 0,C 180,E1 14811.925,E2 14811.925} C_VEL
LIN {X 0,Y 353.126,Z 446.485,A -85,B 0,C 180,E1 14809.47,E2 14809.47} C_VEL
LIN {X 0,Y 349.979,Z 442.331,A -85,B 0,C 180,E1 14807.227,E2 14807.227} C_VEL
LIN {X 0,Y 346.294,Z 439.725,A -85,B 0,C 180,E1 14804.892,E2 14804.892} C_VEL
LIN {X 0,Y 343.02,Z 435.592,A -85,B 0,C 180,E1 14802.733,E2 14802.733} C_VEL
LIN {X 0,Y 338.489,Z 431.902,A -85,B 0,C 180,E1 14799.963,E2 14799.963} C_VEL
LIN {X 0,Y 335.585,Z 428.134,A -85,B 0,C 180,E1 14798.136,E2 14798.136} C_VEL
LIN {X 0,Y 331.971,Z 425.318,A -85,B 0,C 180,E1 14796.061,E2 14796.061} C_VEL
LIN {X 0,Y 328.698,Z 421.265,A -85,B 0,C 180,E1 14794.234,E2 14794.234} C_VEL
LIN {X 0,Y 324.842,Z 418.425,A -85,B 0,C 180,E1 14792.371,E2 14792.371} C_VEL
LIN {X 0,Y 321.093,Z 413.971,A -85,B 0,C 180,E1 14790.594,E2 14790.594} C_VEL
LIN {X 0,Y 317.47,Z 410.98,A -85,B 0,C 180,E1 14789.054,E2 14789.054} C_VEL
LIN {X 0,Y 314.439,Z 407.082,A -85,B 0,C 180,E1 14787.754,E2 14787.754} C_VEL
LIN {X 0,Y 310.861,Z 403.842,A -85,B 0,C 180,E1 14786.288,E2 14786.288} C_VEL
LIN {X 0,Y 308.935,Z 400.729,A -85,B 0,C 180,E1 14785.383,E2 14785.383} C_VEL
LIN {X 0,Y 305.719,Z 398.033,A -85,B 0,C 180,E1 14783.914,E2 14783.914} C_VEL
LIN {X 0,Y 303.571,Z 394.446,A -85,B 0,C 180,E1 14782.758,E2 14782.758} C_VEL
LIN {X 0,Y 299.991,Z 391.927,A -85,B 0,C 180,E1 14780.883,E2 14780.883} C_VEL
LIN {X 0,Y 298.406,Z 388.649,A -85,B 0,C 180,E1 14779.694,E2 14779.694} C_VEL
LIN {X 0,Y 298.234,Z 387.86,A -85,B 0,C 180,E1 14778.765,E2 14778.765} C_VEL
LIN {X 0,Y 298.243,Z 387.81,A -85,B 0,C 180,E1 14774.156,E2 14774.156} C_VEL
LIN {X 0,Y 298.25,Z 387.757,A -85,B 0,C 180,E1 14769.64,E2 14769.64} C_VEL
LIN {X 0,Y 298.244,Z 387.829,A -85,B 0,C 180,E1 14765.185,E2 14765.185} C_VEL
LIN {X 0,Y 298.22,Z 387.763,A -85,B 0,C 180,E1 14760.568,E2 14760.568} C_VEL
LIN {X 0,Y 298.234,Z 387.82,A -85,B 0,C 180,E1 14758.2,E2 14758.2} C_VEL
LIN {X 0,Y 297.402,Z 387.948,A -85,B 0,C 180,E1 14756.825,E2 14756.825} C_VEL
LIN {X 0,Y 293.769,Z 388.362,A -85,B 0,C 180,E1 14754.546,E2 14754.546} C_VEL
LIN {X 0,Y 290.674,Z 388.712,A -85,B 0,C 180,E1 14752.307,E2 14752.307} C_VEL
LIN {X 0,Y 290.317,Z 388.767,A -85,B 0,C 180,E1 14751.424,E2 14751.424} C_VEL
LIN {X 0,Y 290.308,Z 388.825,A -85,B 0,C 180,E1 14746.853,E2 14746.853} C_VEL
LIN {X 0,Y 290.484,Z 389.709,A -85,B 0,C 180,E1 14745.643,E2 14745.643} C_VEL
LIN {X 0,Y 292.276,Z 393.124,A -85,B 0,C 180,E1 14743.905,E2 14743.905} C_VEL
LIN {X 0,Y 295.603,Z 395.394,A -85,B 0,C 180,E1 14741.658,E2 14741.658} C_VEL
LIN {X 0,Y 296.462,Z 396.331,A -85,B 0,C 180,E1 14741.101,E2 14741.101} C_VEL
LIN {X 0,Y 298.447,Z 399.621,A -85,B 0,C 180,E1 14739.807,E2 14739.807} C_VEL
LIN {X 0,Y 301.864,Z 402.332,A -85,B 0,C 180,E1 14737.961,E2 14737.961} C_VEL
LIN {X 0,Y 304.256,Z 406.109,A -85,B 0,C 180,E1 14736.665,E2 14736.665} C_VEL
LIN {X 0,Y 307.236,Z 408.82,A -85,B 0,C 180,E1 14735.273,E2 14735.273} C_VEL
LIN {X 0,Y 310.446,Z 413.064,A -85,B 0,C 180,E1 14733.81,E2 14733.81} C_VEL
LIN {X 0,Y 312.16,Z 414.881,A -85,B 0,C 180,E1 14733.094,E2 14733.094} C_VEL
LIN {X 0,Y 315.756,Z 419.381,A -85,B 0,C 180,E1 14731.635,E2 14731.635} C_VEL
LIN {X 0,Y 321.275,Z 426.681,A -85,B 0,C 180,E1 14729.562,E2 14729.562} C_VEL
LIN {X 0,Y 329.366,Z 439.394,A -85,B 0,C 180,E1 14726.768,E2 14726.768} C_VEL
LIN {X 0,Y 336.573,Z 451.559,A -85,B 0,C 180,E1 14724.515,E2 14724.515} C_VEL
LIN {X 0,Y 344.052,Z 465.245,A -85,B 0,C 180,E1 14722.358,E2 14722.358} C_VEL
LIN {X 0,Y 350.942,Z 479.155,A -85,B 0,C 180,E1 14720.494,E2 14720.494} C_VEL
LIN {X 0,Y 341.927,Z 644.859,A -85,B 0,C 180,E1 14717.031,E2 14717.031} C_VEL
LIN {X 0,Y 339.664,Z 666.141,A -85,B 0,C 180,E1 14716.38,E2 14716.38} C_VEL
LIN {X 0,Y 336.754,Z 684.664,A -85,B 0,C 180,E1 14715.565,E2 14715.565} C_VEL
LIN {X 0,Y 333.653,Z 700.898,A -85,B 0,C 180,E1 14714.644,E2 14714.644} C_VEL
LIN {X 0,Y 329.464,Z 719.727,A -85,B 0,C 180,E1 14713.302,E2 14713.302} C_VEL
LIN {X 0,Y 324.757,Z 737.477,A -85,B 0,C 180,E1 14711.682,E2 14711.682} C_VEL
LIN {X 0,Y 320.355,Z 752.62,A -85,B 0,C 180,E1 14710.01,E2 14710.01} C_VEL
LIN {X 0,Y 315.063,Z 769.469,A -85,B 0,C 180,E1 14707.768,E2 14707.768} C_VEL
LIN {X 0,Y 310.061,Z 784.111,A -85,B 0,C 180,E1 14705.367,E2 14705.367} C_VEL
LIN {X 0,Y 305.911,Z 795.932,A -85,B 0,C 180,E1 14703.08,E2 14703.08} C_VEL
LIN {X 0,Y 301.292,Z 809.082,A -85,B 0,C 180,E1 14700.072,E2 14700.072} C_VEL
LIN {X 0,Y 297.187,Z 820.675,A -85,B 0,C 180,E1 14696.796,E2 14696.796} C_VEL
LIN {X 0,Y 294.266,Z 829.429,A -85,B 0,C 180,E1 14693.849,E2 14693.849} C_VEL
LIN {X 0,Y 291.601,Z 838.322,A -85,B 0,C 180,E1 14690.261,E2 14690.261} C_VEL
LIN {X 0,Y 289.623,Z 845.978,A -85,B 0,C 180,E1 14686.298,E2 14686.298} C_VEL
LIN {X 0,Y 288.638,Z 850.979,A -85,B 0,C 180,E1 14683.012,E2 14683.012} C_VEL
LIN {X 0,Y 288.129,Z 854.973,A -85,B 0,C 180,E1 14679.588,E2 14679.588} C_VEL
LIN {X 0,Y 287.957,Z 858.224,A -85,B 0,C 180,E1 14675.379,E2 14675.379} C_VEL
LIN {X 0,Y 287.97,Z 859.466,A -85,B 0,C 180,E1 14671.99,E2 14671.99} C_VEL
LIN {X 0,Y 287.98,Z 859.585,A -85,B 0,C 180,E1 14668.806,E2 14668.806} C_VEL
LIN {X 0,Y 287.953,Z 858.672,A -85,B 0,C 180,E1 14665.619,E2 14665.619} C_VEL
LIN {X 0,Y 288.011,Z 856.72,A -85,B 0,C 180,E1 14662.42,E2 14662.42} C_VEL
LIN {X 0,Y 288.342,Z 853.08,A -85,B 0,C 180,E1 14658.601,E2 14658.601} C_VEL
LIN {X 0,Y 289.307,Z 847.42,A -85,B 0,C 180,E1 14654.567,E2 14654.567} C_VEL
LIN {X 0,Y 290.785,Z 841.204,A -85,B 0,C 180,E1 14651.143,E2 14651.143} C_VEL
LIN {X 0,Y 293.285,Z 832.665,A -85,B 0,C 180,E1 14647.342,E2 14647.342} C_VEL
LIN {X 0,Y 296.61,Z 822.365,A -85,B 0,C 180,E1 14643.735,E2 14643.735} C_VEL
LIN {X 0,Y 300.068,Z 812.393,A -85,B 0,C 180,E1 14640.82,E2 14640.82} C_VEL
LIN {X 0,Y 304.698,Z 799.503,A -85,B 0,C 180,E1 14637.665,E2 14637.665} C_VEL
LIN {X 0,Y 309.536,Z 785.613,A -85,B 0,C 180,E1 14634.904,E2 14634.904} C_VEL
LIN {X 0,Y 313.9,Z 772.84,A -85,B 0,C 180,E1 14632.758,E2 14632.758} C_VEL
LIN {X 0,Y 319.106,Z 756.889,A -85,B 0,C 180,E1 14630.503,E2 14630.503} C_VEL
LIN {X 0,Y 324.034,Z 740.055,A -85,B 0,C 180,E1 14628.581,E2 14628.581} C_VEL
LIN {X 0,Y 328.011,Z 725.271,A -85,B 0,C 180,E1 14627.177,E2 14627.177} C_VEL
LIN {X 0,Y 332.401,Z 706.999,A -85,B 0,C 180,E1 14625.747,E2 14625.747} C_VEL
LIN {X 0,Y 336.293,Z 687.27,A -85,B 0,C 180,E1 14624.567,E2 14624.567} C_VEL
LIN {X 0,Y 339.012,Z 670.49,A -85,B 0,C 180,E1 14623.795,E2 14623.795} C_VEL
LIN {X 0,Y 341.526,Z 650.232,A -85,B 0,C 180,E1 14623.102,E2 14623.102} C_VEL
LIN {X 0,Y 343.603,Z 616.231,A -85,B 0,C 180,E1 14622.342,E2 14622.342} C_VEL
LIN {X 0,Y 350.816,Z 478.744,A -85,B 0,C 180,E1 14619.468,E2 14619.468} C_VEL
LIN {X 0,Y 342.188,Z 461.692,A -85,B 0,C 180,E1 14617.119,E2 14617.119} C_VEL
LIN {X 0,Y 333.935,Z 446.914,A -85,B 0,C 180,E1 14614.679,E2 14614.679} C_VEL
LIN {X 0,Y 326.565,Z 434.904,A -85,B 0,C 180,E1 14612.301,E2 14612.301} C_VEL
LIN {X 0,Y 319.737,Z 424.505,A -85,B 0,C 180,E1 14609.874,E2 14609.874} C_VEL
LIN {X 0,Y 315.432,Z 419.075,A -85,B 0,C 180,E1 14608.242,E2 14608.242} C_VEL
LIN {X 0,Y 311.873,Z 414.385,A -85,B 0,C 180,E1 14606.779,E2 14606.779} C_VEL
LIN {X 0,Y 308.032,Z 410.154,A -85,B 0,C 180,E1 14605.115,E2 14605.115} C_VEL
LIN {X 0,Y 306.685,Z 408.122,A -85,B 0,C 180,E1 14604.466,E2 14604.466} C_VEL
LIN {X 0,Y 303.387,Z 405.038,A -85,B 0,C 180,E1 14602.892,E2 14602.892} C_VEL
LIN {X 0,Y 301.443,Z 401.894,A -85,B 0,C 180,E1 14601.815,E2 14601.815} C_VEL
LIN {X 0,Y 298.141,Z 399.266,A -85,B 0,C 180,E1 14600.011,E2 14600.011} C_VEL
LIN {X 0,Y 295.91,Z 395.505,A -85,B 0,C 180,E1 14598.526,E2 14598.526} C_VEL
LIN {X 0,Y 292.527,Z 393.387,A -85,B 0,C 180,E1 14596.284,E2 14596.284} C_VEL
LIN {X 0,Y 290.774,Z 390.582,A -85,B 0,C 180,E1 14594.8,E2 14594.8} C_VEL
LIN {X 0,Y 290.335,Z 389.096,A -85,B 0,C 180,E1 14593.754,E2 14593.754} C_VEL
LIN {X 0,Y 290.312,Z 388.824,A -85,B 0,C 180,E1 14590.325,E2 14590.325} C_VEL
LIN {X 0,Y 290.284,Z 388.749,A -85,B 0,C 180,E1 14585.741,E2 14585.741} C_VEL
LIN {X 0,Y 290.292,Z 388.785,A -85,B 0,C 180,E1 14581.193,E2 14581.193} C_VEL
LIN {X 0,Y 290.304,Z 388.759,A -85,B 0,C 180,E1 14576.652,E2 14576.652} C_VEL
LIN {X 0,Y 290.324,Z 388.758,A -85,B 0,C 180,E1 14572.29,E2 14572.29} C_VEL
LIN {X 0,Y 290.294,Z 388.791,A -85,B 0,C 180,E1 14567.679,E2 14567.679} C_VEL
LIN {X 0,Y 290.358,Z 389.215,A -85,B 0,C 180,E1 14565.655,E2 14565.655} C_VEL
LIN {X 0,Y 290.929,Z 391.04,A -85,B 0,C 180,E1 14564.614,E2 14564.614} C_VEL
LIN {X 0,Y 293.145,Z 393.944,A -85,B 0,C 180,E1 14562.851,E2 14562.851} C_VEL
LIN {X 0,Y 296.373,Z 396.061,A -85,B 0,C 180,E1 14560.755,E2 14560.755} C_VEL
LIN {X 0,Y 298.249,Z 399.475,A -85,B 0,C 180,E1 14559.503,E2 14559.503} C_VEL
LIN {X 0,Y 301.984,Z 402.527,A -85,B 0,C 180,E1 14557.478,E2 14557.478} C_VEL
LIN {X 0,Y 304.398,Z 406.229,A -85,B 0,C 180,E1 14556.181,E2 14556.181} C_VEL
LIN {X 0,Y 307.102,Z 408.662,A -85,B 0,C 180,E1 14554.919,E2 14554.919} C_VEL
LIN {X 0,Y 310.001,Z 412.665,A -85,B 0,C 180,E1 14553.581,E2 14553.581} C_VEL
LIN {X 0,Y 313.082,Z 415.431,A -85,B 0,C 180,E1 14552.322,E2 14552.322} C_VEL
LIN {X 0,Y 316.638,Z 419.648,A -85,B 0,C 180,E1 14550.811,E2 14550.811} C_VEL
LIN {X 0,Y 319.977,Z 422.413,A -85,B 0,C 180,E1 14549.392,E2 14549.392} C_VEL
LIN {X 0,Y 323.599,Z 426.511,A -85,B 0,C 180,E1 14547.699,E2 14547.699} C_VEL
LIN {X 0,Y 327.629,Z 429.649,A -85,B 0,C 180,E1 14545.745,E2 14545.745} C_VEL
LIN {X 0,Y 331.101,Z 433.662,A -85,B 0,C 180,E1 14543.829,E2 14543.829} C_VEL
LIN {X 0,Y 334.656,Z 436.463,A -85,B 0,C 180,E1 14541.79,E2 14541.79} C_VEL
LIN {X 0,Y 337.798,Z 440.377,A -85,B 0,C 180,E1 14539.828,E2 14539.828} C_VEL
LIN {X 0,Y 341.71,Z 443.588,A -85,B 0,C 180,E1 14537.432,E2 14537.432} C_VEL
LIN {X 0,Y 345.326,Z 447.887,A -85,B 0,C 180,E1 14535.065,E2 14535.065} C_VEL
LIN {X 0,Y 348.785,Z 450.486,A -85,B 0,C 180,E1 14532.863,E2 14532.863} C_VEL
LIN {X 0,Y 352.18,Z 454.633,A -85,B 0,C 180,E1 14530.475,E2 14530.475} C_VEL
LIN {X 0,Y 356.139,Z 457.65,A -85,B 0,C 180,E1 14527.735,E2 14527.735} C_VEL
LIN {X 0,Y 359.483,Z 461.702,A -85,B 0,C 180,E1 14525.151,E2 14525.151} C_VEL
LIN {X 0,Y 362.902,Z 464.069,A -85,B 0,C 180,E1 14522.552,E2 14522.552} C_VEL
LIN {X 0,Y 363.845,Z 464.973,A -85,B 0,C 180,E1 14521.749,E2 14521.749} C_VEL
LIN {X 0,Y 366.49,Z 468.363,A -85,B 0,C 180,E1 14519.41,E2 14519.41} C_VEL
LIN {X 0,Y 369.463,Z 470.745,A -85,B 0,C 180,E1 14516.694,E2 14516.694} C_VEL
LIN {X 0,Y 371.691,Z 472.115,A -85,B 0,C 180,E1 14514.565,E2 14514.565} C_VEL
LIN {X 0,Y 373.814,Z 475.193,A -85,B 0,C 180,E1 14512.156,E2 14512.156} C_VEL
LIN {X 0,Y 376.422,Z 477.524,A -85,B 0,C 180,E1 14509.016,E2 14509.016} C_VEL
LIN {X 0,Y 378.909,Z 478.763,A -85,B 0,C 180,E1 14505.614,E2 14505.614} C_VEL
LIN {X 0,Y 380.141,Z 479.888,A -85,B 0,C 180,E1 14503.538,E2 14503.538} C_VEL
LIN {X 0,Y 381.517,Z 482.161,A -85,B 0,C 180,E1 14500.571,E2 14500.571} C_VEL
LIN {X 0,Y 382.659,Z 483.515,A -85,B 0,C 180,E1 14497.356,E2 14497.356} C_VEL
LIN {X 0,Y 383.466,Z 484.221,A -85,B 0,C 180,E1 14494.037,E2 14494.037} C_VEL
LIN {X 0,Y 383.788,Z 484.461,A -85,B 0,C 180,E1 14490.746,E2 14490.746} C_VEL
LIN {X 0,Y 383.665,Z 484.364,A -85,B 0,C 180,E1 14487.311,E2 14487.311} C_VEL
LIN {X 0,Y 383.06,Z 483.856,A -85,B 0,C 180,E1 14484.007,E2 14484.007} C_VEL
LIN {X 0,Y 381.99,Z 482.774,A -85,B 0,C 180,E1 14480.614,E2 14480.614} C_VEL
LIN {X 0,Y 380.703,Z 480.848,A -85,B 0,C 180,E1 14477.564,E2 14477.564} C_VEL
LIN {X 0,Y 379.326,Z 478.968,A -85,B 0,C 180,E1 14475.03,E2 14475.03} C_VEL
LIN {X 0,Y 376.882,Z 477.82,A -85,B 0,C 180,E1 14471.597,E2 14471.597} C_VEL
LIN {X 0,Y 374.245,Z 475.682,A -85,B 0,C 180,E1 14468.366,E2 14468.366} C_VEL
LIN {X 0,Y 371.914,Z 472.491,A -85,B 0,C 180,E1 14465.67,E2 14465.67} C_VEL
LIN {X 0,Y 371.063,Z 471.556,A -85,B 0,C 180,E1 14464.803,E2 14464.803} C_VEL
LIN {X 0,Y 367.741,Z 469.542,A -85,B 0,C 180,E1 14461.733,E2 14461.733} C_VEL
LIN {X 0,Y 364.785,Z 466.349,A -85,B 0,C 180,E1 14459.063,E2 14459.063} C_VEL
LIN {X 0,Y 363.182,Z 464.213,A -85,B 0,C 180,E1 14457.673,E2 14457.673} C_VEL
LIN {X 0,Y 359.751,Z 461.961,A -85,B 0,C 180,E1 14455.056,E2 14455.056} C_VEL
LIN {X 0,Y 356.279,Z 457.857,A -85,B 0,C 180,E1 14452.366,E2 14452.366} C_VEL
LIN {X 0,Y 355.069,Z 456.737,A -85,B 0,C 180,E1 14451.515,E2 14451.515} C_VEL
LIN {X 0,Y 351.345,Z 453.793,A -85,B 0,C 180,E1 14448.934,E2 14448.934} C_VEL
LIN {X 0,Y 348.278,Z 449.916,A -85,B 0,C 180,E1 14446.804,E2 14446.804} C_VEL
LIN {X 0,Y 344.751,Z 447.329,A -85,B 0,C 180,E1 14444.562,E2 14444.562} C_VEL
LIN {X 0,Y 341.032,Z 442.824,A -85,B 0,C 180,E1 14442.12,E2 14442.12} C_VEL
LIN {X 0,Y 336.892,Z 439.502,A -85,B 0,C 180,E1 14439.637,E2 14439.637} C_VEL
LIN {X 0,Y 334.024,Z 435.834,A -85,B 0,C 180,E1 14437.841,E2 14437.841} C_VEL
LIN {X 0,Y 330.325,Z 432.914,A -85,B 0,C 180,E1 14435.734,E2 14435.734} C_VEL
LIN {X 0,Y 326.791,Z 428.815,A -85,B 0,C 180,E1 14433.826,E2 14433.826} C_VEL
LIN {X 0,Y 322.708,Z 425.674,A -85,B 0,C 180,E1 14431.887,E2 14431.887} C_VEL
LIN {X 0,Y 319.041,Z 421.448,A -85,B 0,C 180,E1 14430.187,E2 14430.187} C_VEL
LIN {X 0,Y 315.155,Z 418.14,A -85,B 0,C 180,E1 14428.561,E2 14428.561} C_VEL
LIN {X 0,Y 312.056,Z 414.356,A -85,B 0,C 180,E1 14427.259,E2 14427.259} C_VEL
LIN {X 0,Y 308.455,Z 410.859,A -85,B 0,C 180,E1 14425.734,E2 14425.734} C_VEL
LIN {X 0,Y 306.644,Z 408.074,A -85,B 0,C 180,E1 14424.863,E2 14424.863} C_VEL
LIN {X 0,Y 303.439,Z 405.06,A -85,B 0,C 180,E1 14423.332,E2 14423.332} C_VEL
LIN {X 0,Y 301.755,Z 402.075,A -85,B 0,C 180,E1 14422.388,E2 14422.388} C_VEL
LIN {X 0,Y 298.249,Z 399.475,A -85,B 0,C 180,E1 14420.497,E2 14420.497} C_VEL
LIN {X 0,Y 296.016,Z 395.645,A -85,B 0,C 180,E1 14419.013,E2 14419.013} C_VEL
LIN {X 0,Y 292.124,Z 392.937,A -85,B 0,C 180,E1 14416.392,E2 14416.392} C_VEL
LIN {X 0,Y 290.394,Z 389.424,A -85,B 0,C 180,E1 14414.547,E2 14414.547} C_VEL
LIN {X 0,Y 290.308,Z 388.843,A -85,B 0,C 180,E1 14413.332,E2 14413.332} C_VEL
LIN {X 0,Y 290.283,Z 388.75,A -85,B 0,C 180,E1 14408.69,E2 14408.69} C_VEL
LIN {X 0,Y 290.295,Z 388.779,A -85,B 0,C 180,E1 14404.139,E2 14404.139} C_VEL
LIN {X 0,Y 290.322,Z 388.761,A -85,B 0,C 180,E1 14399.597,E2 14399.597} C_VEL
LIN {X 0,Y 290.298,Z 388.756,A -85,B 0,C 180,E1 14395.052,E2 14395.052} C_VEL
LIN {X 0,Y 290.317,Z 388.767,A -85,B 0,C 180,E1 14391.424,E2 14391.424} C_VEL
LIN {X 0,Y 290.003,Z 389.775,A -85,B 0,C 180,E1 14389.905,E2 14389.905} C_VEL
LIN {X 0,Y 289.228,Z 393.462,A -85,B 0,C 180,E1 14387.82,E2 14387.82} C_VEL
LIN {X 0,Y 289.451,Z 398.458,A -85,B 0,C 180,E1 14385.563,E2 14385.563} C_VEL
LIN {X 0,Y 290.189,Z 400.024,A -85,B 0,C 180,E1 14384.739,E2 14384.739} C_VEL
LIN {X 0,Y 293.478,Z 402.897,A -85,B 0,C 180,E1 14382.341,E2 14382.341} C_VEL
LIN {X 0,Y 294.56,Z 403.662,A -85,B 0,C 180,E1 14381.642,E2 14381.642} C_VEL
LIN {X 0,Y 296.714,Z 407.163,A -85,B 0,C 180,E1 14380.197,E2 14380.197} C_VEL
LIN {X 0,Y 299.955,Z 410.027,A -85,B 0,C 180,E1 14378.38,E2 14378.38} C_VEL
LIN {X 0,Y 302.766,Z 414.029,A -85,B 0,C 180,E1 14376.852,E2 14376.852} C_VEL
LIN {X 0,Y 305.144,Z 416.319,A -85,B 0,C 180,E1 14375.711,E2 14375.711} C_VEL
LIN {X 0,Y 308.509,Z 420.612,A -85,B 0,C 180,E1 14374.15,E2 14374.15} C_VEL
LIN {X 0,Y 310.171,Z 422.691,A -85,B 0,C 180,E1 14373.424,E2 14373.424} C_VEL
LIN {X 0,Y 314.556,Z 428.281,A -85,B 0,C 180,E1 14371.62,E2 14371.62} C_VEL
LIN {X 0,Y 318.41,Z 433.441,A -85,B 0,C 180,E1 14370.144,E2 14370.144} C_VEL
LIN {X 0,Y 326.054,Z 445.692,A -85,B 0,C 180,E1 14367.408,E2 14367.408} C_VEL
LIN {X 0,Y 333.362,Z 458.288,A -85,B 0,C 180,E1 14365.043,E2 14365.043} C_VEL
LIN {X 0,Y 341.479,Z 473.613,A -85,B 0,C 180,E1 14362.633,E2 14362.633} C_VEL
LIN {X 0,Y 345.678,Z 482.61,A -85,B 0,C 180,E1 14361.444,E2 14361.444} C_VEL
LIN {X 0,Y 336.515,Z 644.536,A -85,B 0,C 180,E1 14358.033,E2 14358.033} C_VEL
LIN {X 0,Y 334.21,Z 665.675,A -85,B 0,C 180,E1 14357.387,E2 14357.387} C_VEL
LIN {X 0,Y 331.169,Z 684.426,A -85,B 0,C 180,E1 14356.56,E2 14356.56} C_VEL
LIN {X 0,Y 327.963,Z 700.66,A -85,B 0,C 180,E1 14355.635,E2 14355.635} C_VEL
LIN {X 0,Y 323.626,Z 719.488,A -85,B 0,C 180,E1 14354.284,E2 14354.284} C_VEL
LIN {X 0,Y 318.745,Z 737.238,A -85,B 0,C 180,E1 14352.652,E2 14352.652} C_VEL
LIN {X 0,Y 314.41,Z 751.596,A -85,B 0,C 180,E1 14351.059,E2 14351.059} C_VEL
LIN {X 0,Y 309.053,Z 768.052,A -85,B 0,C 180,E1 14348.874,E2 14348.874} C_VEL
LIN {X 0,Y 303.612,Z 783.368,A -85,B 0,C 180,E1 14346.353,E2 14346.353} C_VEL
LIN {X 0,Y 299.075,Z 795.689,A -85,B 0,C 180,E1 14343.938,E2 14343.938} C_VEL
LIN {X 0,Y 294.213,Z 808.839,A -85,B 0,C 180,E1 14340.874,E2 14340.874} C_VEL
LIN {X 0,Y 289.872,Z 820.432,A -85,B 0,C 180,E1 14337.529,E2 14337.529} C_VEL
LIN {X 0,Y 286.722,Z 829.326,A -85,B 0,C 180,E1 14334.461,E2 14334.461} C_VEL
LIN {X 0,Y 283.788,Z 838.538,A -85,B 0,C 180,E1 14330.629,E2 14330.629} C_VEL
LIN {X 0,Y 281.718,Z 846.013,A -85,B 0,C 180,E1 14326.594,E2 14326.594} C_VEL
LIN {X 0,Y 280.668,Z 851.011,A -85,B 0,C 180,E1 14323.179,E2 14323.179} C_VEL
LIN {X 0,Y 280.098,Z 855.364,A -85,B 0,C 180,E1 14319.243,E2 14319.243} C_VEL
LIN {X 0,Y 279.957,Z 858.166,A -85,B 0,C 180,E1 14315.122,E2 14315.122} C_VEL
LIN {X 0,Y 279.975,Z 859.259,A -85,B 0,C 180,E1 14311.842,E2 14311.842} C_VEL
LIN {X 0,Y 279.983,Z 859.349,A -85,B 0,C 180,E1 14308.772,E2 14308.772} C_VEL
LIN {X 0,Y 279.956,Z 858.435,A -85,B 0,C 180,E1 14305.494,E2 14305.494} C_VEL
LIN {X 0,Y 280.016,Z 856.482,A -85,B 0,C 180,E1 14302.202,E2 14302.202} C_VEL
LIN {X 0,Y 280.391,Z 852.84,A -85,B 0,C 180,E1 14298.273,E2 14298.273} C_VEL
LIN {X 0,Y 281.448,Z 847.179,A -85,B 0,C 180,E1 14294.125,E2 14294.125} C_VEL
LIN {X 0,Y 283.042,Z 840.962,A -85,B 0,C 180,E1 14290.607,E2 14290.607} C_VEL
LIN {X 0,Y 285.721,Z 832.422,A -85,B 0,C 180,E1 14286.708,E2 14286.708} C_VEL
LIN {X 0,Y 289.198,Z 822.296,A -85,B 0,C 180,E1 14283.07,E2 14283.07} C_VEL
LIN {X 0,Y 292.834,Z 812.38,A -85,B 0,C 180,E1 14280.1,E2 14280.1} C_VEL
LIN {X 0,Y 297.482,Z 800.11,A -85,B 0,C 180,E1 14277.011,E2 14277.011} C_VEL
LIN {X 0,Y 302.695,Z 785.872,A -85,B 0,C 180,E1 14274.105,E2 14274.105} C_VEL
LIN {X 0,Y 307.24,Z 773.162,A -85,B 0,C 180,E1 14271.926,E2 14271.926} C_VEL
LIN {X 0,Y 312.647,Z 757.314,A -85,B 0,C 180,E1 14269.64,E2 14269.64} C_VEL
LIN {X 0,Y 317.804,Z 740.467,A -85,B 0,C 180,E1 14267.681,E2 14267.681} C_VEL
LIN {X 0,Y 322.118,Z 725.031,A -85,B 0,C 180,E1 14266.198,E2 14266.198} C_VEL
LIN {X 0,Y 326.714,Z 706.581,A -85,B 0,C 180,E1 14264.746,E2 14264.746} C_VEL
LIN {X 0,Y 330.598,Z 687.569,A -85,B 0,C 180,E1 14263.602,E2 14263.602} C_VEL
LIN {X 0,Y 333.434,Z 670.71,A -85,B 0,C 180,E1 14262.817,E2 14262.817} C_VEL
LIN {X 0,Y 335.919,Z 651.497,A -85,B 0,C 180,E1 14262.149,E2 14262.149} C_VEL
LIN {X 0,Y 337.884,Z 622.748,A -85,B 0,C 180,E1 14261.479,E2 14261.479} C_VEL
LIN {X 0,Y 345.641,Z 482.11,A -85,B 0,C 180,E1 14258.532,E2 14258.532} C_VEL
LIN {X 0,Y 337.122,Z 465.214,A -85,B 0,C 180,E1 14256.099,E2 14256.099} C_VEL
LIN {X 0,Y 329.508,Z 451.549,A -85,B 0,C 180,E1 14253.737,E2 14253.737} C_VEL
LIN {X 0,Y 323.255,Z 441.123,A -85,B 0,C 180,E1 14251.626,E2 14251.626} C_VEL
LIN {X 0,Y 317.012,Z 431.407,A -85,B 0,C 180,E1 14249.325,E2 14249.325} C_VEL
LIN {X 0,Y 312.687,Z 425.902,A -85,B 0,C 180,E1 14247.63,E2 14247.63} C_VEL
LIN {X 0,Y 308.709,Z 420.795,A -85,B 0,C 180,E1 14245.935,E2 14245.935} C_VEL
LIN {X 0,Y 305.231,Z 416.468,A -85,B 0,C 180,E1 14244.333,E2 14244.333} C_VEL
LIN {X 0,Y 304.043,Z 415.153,A -85,B 0,C 180,E1 14243.763,E2 14243.763} C_VEL
LIN {X 0,Y 300.813,Z 411.562,A -85,B 0,C 180,E1 14242.12,E2 14242.12} C_VEL
LIN {X 0,Y 299.47,Z 409.416,A -85,B 0,C 180,E1 14241.349,E2 14241.349} C_VEL
LIN {X 0,Y 296.119,Z 406.438,A -85,B 0,C 180,E1 14239.433,E2 14239.433} C_VEL
LIN {X 0,Y 294.368,Z 403.272,A -85,B 0,C 180,E1 14238.217,E2 14238.217} C_VEL
LIN {X 0,Y 290.935,Z 400.945,A -85,B 0,C 180,E1 14235.864,E2 14235.864} C_VEL
LIN {X 0,Y 289.067,Z 397.842,A -85,B 0,C 180,E1 14234.224,E2 14234.224} C_VEL
LIN {X 0,Y 288.02,Z 396.521,A -85,B 0,C 180,E1 14233.253,E2 14233.253} C_VEL
LIN {X 0,Y 284.18,Z 393.939,A -85,B 0,C 180,E1 14229.118,E2 14229.118} C_VEL
LIN {X 0,Y 282.53,Z 390.719,A -85,B 0,C 180,E1 14225.695,E2 14225.695} C_VEL
LIN {X 0,Y 282.378,Z 389.848,A -85,B 0,C 180,E1 14222.241,E2 14222.241} C_VEL
LIN {X 0,Y 282.358,Z 389.84,A -85,B 0,C 180,E1 14217.574,E2 14217.574} C_VEL
LIN {X 0,Y 282.528,Z 390.695,A -85,B 0,C 180,E1 14213.915,E2 14213.915} C_VEL
LIN {X 0,Y 285.422,Z 395.109,A -85,B 0,C 180,E1 14208.901,E2 14208.901} C_VEL
LIN {X 0,Y 288.639,Z 397.065,A -85,B 0,C 180,E1 14205.772,E2 14205.772} C_VEL
LIN {X 0,Y 291.03,Z 401.043,A -85,B 0,C 180,E1 14203.647,E2 14203.647} C_VEL
LIN {X 0,Y 294.533,Z 403.585,A -85,B 0,C 180,E1 14201.248,E2 14201.248} C_VEL
LIN {X 0,Y 296.672,Z 407.196,A -85,B 0,C 180,E1 14199.801,E2 14199.801} C_VEL
LIN {X 0,Y 300.005,Z 410.056,A -85,B 0,C 180,E1 14197.938,E2 14197.938} C_VEL
LIN {X 0,Y 302.731,Z 413.965,A -85,B 0,C 180,E1 14196.455,E2 14196.455} C_VEL
LIN {X 0,Y 305.013,Z 416.185,A -85,B 0,C 180,E1 14195.357,E2 14195.357} C_VEL
LIN {X 0,Y 308.269,Z 420.408,A -85,B 0,C 180,E1 14193.836,E2 14193.836} C_VEL
LIN {X 0,Y 310.799,Z 422.746,A -85,B 0,C 180,E1 14192.777,E2 14192.777} C_VEL
LIN {X 0,Y 314.742,Z 427.212,A -85,B 0,C 180,E1 14191.139,E2 14191.139} C_VEL
LIN {X 0,Y 318.02,Z 429.967,A -85,B 0,C 180,E1 14189.758,E2 14189.758} C_VEL
LIN {X 0,Y 321.977,Z 434.248,A -85,B 0,C 180,E1 14187.937,E2 14187.937} C_VEL
LIN {X 0,Y 325.895,Z 437.295,A -85,B 0,C 180,E1 14186.068,E2 14186.068} C_VEL
LIN {X 0,Y 329.549,Z 441.351,A -85,B 0,C 180,E1 14184.102,E2 14184.102} C_VEL
LIN {X 0,Y 333.157,Z 444.284,A -85,B 0,C 180,E1 14182.043,E2 14182.043} C_VEL
LIN {X 0,Y 336.498,Z 448.257,A -85,B 0,C 180,E1 14179.975,E2 14179.975} C_VEL
LIN {X 0,Y 340.236,Z 451.302,A -85,B 0,C 180,E1 14177.717,E2 14177.717} C_VEL
LIN {X 0,Y 344.083,Z 455.776,A -85,B 0,C 180,E1 14175.2,E2 14175.2} C_VEL
LIN {X 0,Y 347.379,Z 458.29,A -85,B 0,C 180,E1 14173.098,E2 14173.098} C_VEL
LIN {X 0,Y 350.827,Z 462.376,A -85,B 0,C 180,E1 14170.719,E2 14170.719} C_VEL
LIN {X 0,Y 354.727,Z 465.359,A -85,B 0,C 180,E1 14168.005,E2 14168.005} C_VEL
LIN {X 0,Y 358.143,Z 469.425,A -85,B 0,C 180,E1 14165.411,E2 14165.411} C_VEL
LIN {X 0,Y 361.551,Z 471.862,A -85,B 0,C 180,E1 14162.805,E2 14162.805} C_VEL
LIN {X 0,Y 362.582,Z 472.771,A -85,B 0,C 180,E1 14161.968,E2 14161.968} C_VEL
LIN {X 0,Y 365.366,Z 476.274,A -85,B 0,C 180,E1 14159.51,E2 14159.51} C_VEL
LIN {X 0,Y 368.384,Z 478.654,A -85,B 0,C 180,E1 14156.775,E2 14156.775} C_VEL
LIN {X 0,Y 370.53,Z 479.995,A -85,B 0,C 180,E1 14154.724,E2 14154.724} C_VEL
LIN {X 0,Y 372.772,Z 483.137,A -85,B 0,C 180,E1 14152.221,E2 14152.221} C_VEL
LIN {X 0,Y 375.416,Z 485.468,A -85,B 0,C 180,E1 14149.038,E2 14149.038} C_VEL
LIN {X 0,Y 377.901,Z 486.694,A -85,B 0,C 180,E1 14145.656,E2 14145.656} C_VEL
LIN {X 0,Y 379.057,Z 487.712,A -85,B 0,C 180,E1 14143.733,E2 14143.733} C_VEL
LIN {X 0,Y 380.528,Z 490.103,A -85,B 0,C 180,E1 14140.598,E2 14140.598} C_VEL
LIN {X 0,Y 381.676,Z 491.458,A -85,B 0,C 180,E1 14137.375,E2 14137.375} C_VEL
LIN {X 0,Y 382.49,Z 492.161,A -85,B 0,C 180,E1 14134.047,E2 14134.047} C_VEL
LIN {X 0,Y 382.813,Z 492.402,A -85,B 0,C 180,E1 14130.748,E2 14130.748} C_VEL
LIN {X 0,Y 382.69,Z 492.304,A -85,B 0,C 180,E1 14127.305,E2 14127.305} C_VEL
LIN {X 0,Y 382.082,Z 491.796,A -85,B 0,C 180,E1 14123.992,E2 14123.992} C_VEL
LIN {X 0,Y 381.001,Z 490.722,A -85,B 0,C 180,E1 14120.592,E2 14120.592} C_VEL
LIN {X 0,Y 379.707,Z 488.815,A -85,B 0,C 180,E1 14117.531,E2 14117.531} C_VEL
LIN {X 0,Y 378.317,Z 486.9,A -85,B 0,C 180,E1 14114.989,E2 14114.989} C_VEL
LIN {X 0,Y 375.859,Z 485.747,A -85,B 0,C 180,E1 14111.545,E2 14111.545} C_VEL
LIN {X 0,Y 373.199,Z 483.619,A -85,B 0,C 180,E1 14108.302,E2 14108.302} C_VEL
LIN {X 0,Y 370.784,Z 480.431,A -85,B 0,C 180,E1 14105.549,E2 14105.549} C_VEL
LIN {X 0,Y 369.996,Z 479.469,A -85,B 0,C 180,E1 14104.725,E2 14104.725} C_VEL
LIN {X 0,Y 366.681,Z 477.485,A -85,B 0,C 180,E1 14101.677,E2 14101.677} C_VEL
LIN {X 0,Y 363.525,Z 474.156,A -85,B 0,C 180,E1 14098.864,E2 14098.864} C_VEL
LIN {X 0,Y 362.108,Z 472.133,A -85,B 0,C 180,E1 14097.611,E2 14097.611} C_VEL
LIN {X 0,Y 358.595,Z 469.865,A -85,B 0,C 180,E1 14094.945,E2 14094.945} C_VEL
LIN {X 0,Y 354.974,Z 465.717,A -85,B 0,C 180,E1 14092.177,E2 14092.177} C_VEL
LIN {X 0,Y 353.703,Z 464.506,A -85,B 0,C 180,E1 14091.263,E2 14091.263} C_VEL
LIN {X 0,Y 349.958,Z 461.538,A -85,B 0,C 180,E1 14088.697,E2 14088.697} C_VEL
LIN {X 0,Y 346.651,Z 457.567,A -85,B 0,C 180,E1 14086.422,E2 14086.422} C_VEL
LIN {X 0,Y 343.076,Z 454.783,A -85,B 0,C 180,E1 14084.136,E2 14084.136} C_VEL
LIN {X 0,Y 339.343,Z 450.436,A -85,B 0,C 180,E1 14081.738,E2 14081.738} C_VEL
LIN {X 0,Y 335.305,Z 447.102,A -85,B 0,C 180,E1 14079.308,E2 14079.308} C_VEL
LIN {X 0,Y 332.569,Z 443.59,A -85,B 0,C 180,E1 14077.599,E2 14077.599} C_VEL
LIN {X 0,Y 328.649,Z 440.508,A -85,B 0,C 180,E1 14075.408,E2 14075.408} C_VEL
LIN {X 0,Y 324.864,Z 436.344,A -85,B 0,C 180,E1 14073.418,E2 14073.418} C_VEL
LIN {X 0,Y 320.687,Z 433.057,A -85,B 0,C 180,E1 14071.471,E2 14071.471} C_VEL
LIN {X 0,Y 316.941,Z 428.898,A -85,B 0,C 180,E1 14069.782,E2 14069.782} C_VEL
LIN {X 0,Y 312.802,Z 425.304,A -85,B 0,C 180,E1 14068.072,E2 14068.072} C_VEL
LIN {X 0,Y 309.686,Z 421.602,A -85,B 0,C 180,E1 14066.758,E2 14066.758} C_VEL
LIN {X 0,Y 305.987,Z 417.745,A -85,B 0,C 180,E1 14065.127,E2 14065.127} C_VEL
LIN {X 0,Y 304.383,Z 415.38,A -85,B 0,C 180,E1 14064.335,E2 14064.335} C_VEL
LIN {X 0,Y 301.027,Z 411.84,A -85,B 0,C 180,E1 14062.651,E2 14062.651} C_VEL
LIN {X 0,Y 299.778,Z 409.598,A -85,B 0,C 180,E1 14061.924,E2 14061.924} C_VEL
LIN {X 0,Y 296.373,Z 406.84,A -85,B 0,C 180,E1 14060.014,E2 14060.014} C_VEL
LIN {X 0,Y 294.331,Z 403.279,A -85,B 0,C 180,E1 14058.612,E2 14058.612} C_VEL
LIN {X 0,Y 290.665,Z 400.631,A -85,B 0,C 180,E1 14056.066,E2 14056.066} C_VEL
LIN {X 0,Y 288.425,Z 396.836,A -85,B 0,C 180,E1 14054.034,E2 14054.034} C_VEL
LIN {X 0,Y 283.892,Z 393.549,A -85,B 0,C 180,E1 14049.11,E2 14049.11} C_VEL
LIN {X 0,Y 282.508,Z 390.57,A -85,B 0,C 180,E1 14045.882,E2 14045.882} C_VEL
LIN {X 0,Y 282.361,Z 389.835,A -85,B 0,C 180,E1 14042.223,E2 14042.223} C_VEL
LIN {X 0,Y 282.385,Z 389.848,A -85,B 0,C 180,E1 14037.556,E2 14037.556} C_VEL
LIN {X 0,Y 282.53,Z 390.719,A -85,B 0,C 180,E1 14034.305,E2 14034.305} C_VEL
LIN {X 0,Y 285.439,Z 395.152,A -85,B 0,C 180,E1 14029.293,E2 14029.293} C_VEL
LIN {X 0,Y 288.666,Z 397.08,A -85,B 0,C 180,E1 14026.165,E2 14026.165} C_VEL
LIN {X 0,Y 290.189,Z 400.024,A -85,B 0,C 180,E1 14024.739,E2 14024.739} C_VEL
LIN {X 0,Y 292.522,Z 404.512,A -85,B 0,C 180,E1 14022.801,E2 14022.801} C_VEL
LIN {X 0,Y 297.941,Z 417.383,A -85,B 0,C 180,E1 14018.885,E2 14018.885} C_VEL
LIN {X 0,Y 300.929,Z 421.573,A -85,B 0,C 180,E1 14017.22,E2 14017.22} C_VEL
LIN {X 0,Y 302.989,Z 423.636,A -85,B 0,C 180,E1 14016.2,E2 14016.2} C_VEL
LIN {X 0,Y 306.583,Z 428.159,A -85,B 0,C 180,E1 14014.494,E2 14014.494} C_VEL
LIN {X 0,Y 312.219,Z 435.609,A -85,B 0,C 180,E1 14012.066,E2 14012.066} C_VEL
LIN {X 0,Y 315.475,Z 440.013,A -85,B 0,C 180,E1 14010.779,E2 14010.779} C_VEL
LIN {X 0,Y 322.758,Z 451.943,A -85,B 0,C 180,E1 14008.07,E2 14008.07} C_VEL
LIN {X 0,Y 330.484,Z 465.532,A -85,B 0,C 180,E1 14005.486,E2 14005.486} C_VEL
LIN {X 0,Y 338.84,Z 481.952,A -85,B 0,C 180,E1 14002.93,E2 14002.93} C_VEL
LIN {X 0,Y 340.513,Z 486.034,A -85,B 0,C 180,E1 14002.424,E2 14002.424} C_VEL
LIN {X 0,Y 331.193,Z 644.422,A -85,B 0,C 180,E1 13999.063,E2 13999.063} C_VEL
LIN {X 0,Y 328.77,Z 665.781,A -85,B 0,C 180,E1 13998.403,E2 13998.403} C_VEL
LIN {X 0,Y 325.687,Z 684.188,A -85,B 0,C 180,E1 13997.588,E2 13997.588} C_VEL
LIN {X 0,Y 322.375,Z 700.422,A -85,B 0,C 180,E1 13996.66,E2 13996.66} C_VEL
LIN {X 0,Y 317.887,Z 719.249,A -85,B 0,C 180,E1 13995.302,E2 13995.302} C_VEL
LIN {X 0,Y 312.829,Z 736.998,A -85,B 0,C 180,E1 13993.658,E2 13993.658} C_VEL
LIN {X 0,Y 308.244,Z 751.606,A -85,B 0,C 180,E1 13992.021,E2 13992.021} C_VEL
LIN {X 0,Y 302.532,Z 768.416,A -85,B 0,C 180,E1 13989.754,E2 13989.754} C_VEL
LIN {X 0,Y 296.871,Z 783.627,A -85,B 0,C 180,E1 13987.195,E2 13987.195} C_VEL
LIN {X 0,Y 292.232,Z 795.651,A -85,B 0,C 180,E1 13984.791,E2 13984.791} C_VEL
LIN {X 0,Y 287.192,Z 808.597,A -85,B 0,C 180,E1 13981.715,E2 13981.715} C_VEL
LIN {X 0,Y 282.606,Z 820.189,A -85,B 0,C 180,E1 13978.299,E2 13978.299} C_VEL
LIN {X 0,Y 279.314,Z 828.944,A -85,B 0,C 180,E1 13975.212,E2 13975.212} C_VEL
LIN {X 0,Y 276.266,Z 837.837,A -85,B 0,C 180,E1 13971.44,E2 13971.44} C_VEL
LIN {X 0,Y 274.032,Z 845.257,A -85,B 0,C 180,E1 13967.409,E2 13967.409} C_VEL
LIN {X 0,Y 272.792,Z 850.553,A -85,B 0,C 180,E1 13963.739,E2 13963.739} C_VEL
LIN {X 0,Y 272.161,Z 854.705,A -85,B 0,C 180,E1 13959.943,E2 13959.943} C_VEL
LIN {X 0,Y 271.961,Z 857.749,A -85,B 0,C 180,E1 13955.697,E2 13955.697} C_VEL
LIN {X 0,Y 271.975,Z 858.993,A -85,B 0,C 180,E1 13952.107,E2 13952.107} C_VEL
LIN {X 0,Y 271.986,Z 859.112,A -85,B 0,C 180,E1 13948.736,E2 13948.736} C_VEL
LIN {X 0,Y 271.958,Z 858.198,A -85,B 0,C 180,E1 13945.361,E2 13945.361} C_VEL
LIN {X 0,Y 272.024,Z 856.244,A -85,B 0,C 180,E1 13941.971,E2 13941.971} C_VEL
LIN {X 0,Y 272.444,Z 852.6,A -85,B 0,C 180,E1 13937.926,E2 13937.926} C_VEL
LIN {X 0,Y 273.602,Z 846.938,A -85,B 0,C 180,E1 13933.657,E2 13933.657} C_VEL
LIN {X 0,Y 275.324,Z 840.719,A -85,B 0,C 180,E1 13930.04,E2 13930.04} C_VEL
LIN {X 0,Y 278.194,Z 832.179,A -85,B 0,C 180,E1 13926.039,E2 13926.039} C_VEL
LIN {X 0,Y 281.893,Z 822.054,A -85,B 0,C 180,E1 13922.313,E2 13922.313} C_VEL
LIN {X 0,Y 285.74,Z 812.137,A -85,B 0,C 180,E1 13919.278,E2 13919.278} C_VEL
LIN {X 0,Y 290.633,Z 799.867,A -85,B 0,C 180,E1 13916.13,E2 13916.13} C_VEL
LIN {X 0,Y 296.156,Z 785.497,A -85,B 0,C 180,E1 13913.152,E2 13913.152} C_VEL
LIN {X 0,Y 300.853,Z 772.92,A -85,B 0,C 180,E1 13910.967,E2 13910.967} C_VEL
LIN {X 0,Y 306.26,Z 757.706,A -85,B 0,C 180,E1 13908.742,E2 13908.742} C_VEL
LIN {X 0,Y 311.851,Z 740.227,A -85,B 0,C 180,E1 13906.677,E2 13906.677} C_VEL
LIN {X 0,Y 316.326,Z 724.792,A -85,B 0,C 180,E1 13905.183,E2 13905.183} C_VEL
LIN {X 0,Y 321.039,Z 706.522,A -85,B 0,C 180,E1 13903.736,E2 13903.736} C_VEL
LIN {X 0,Y 325.104,Z 687.312,A -85,B 0,C 180,E1 13902.574,E2 13902.574} C_VEL
LIN {X 0,Y 328.01,Z 670.587,A -85,B 0,C 180,E1 13901.793,E2 13901.793} C_VEL
LIN {X 0,Y 330.534,Z 651.703,A -85,B 0,C 180,E1 13901.132,E2 13901.132} C_VEL
LIN {X 0,Y 332.558,Z 623.658,A -85,B 0,C 180,E1 13900.467,E2 13900.467} C_VEL
LIN {X 0,Y 340.423,Z 485.36,A -85,B 0,C 180,E1 13897.534,E2 13897.534} C_VEL
LIN {X 0,Y 332.112,Z 468.579,A -85,B 0,C 180,E1 13895.029,E2 13895.029} C_VEL
LIN {X 0,Y 324.381,Z 454.666,A -85,B 0,C 180,E1 13892.493,E2 13892.493} C_VEL
LIN {X 0,Y 317.927,Z 443.898,A -85,B 0,C 180,E1 13890.166,E2 13890.166} C_VEL
LIN {X 0,Y 314.102,Z 438.056,A -85,B 0,C 180,E1 13888.684,E2 13888.684} C_VEL
LIN {X 0,Y 309.981,Z 432.704,A -85,B 0,C 180,E1 13887.007,E2 13887.007} C_VEL
LIN {X 0,Y 306.192,Z 427.785,A -85,B 0,C 180,E1 13885.334,E2 13885.334} C_VEL
LIN {X 0,Y 302.186,Z 422.699,A -85,B 0,C 180,E1 13883.401,E2 13883.401} C_VEL
LIN {X 0,Y 298.764,Z 418.829,A -85,B 0,C 180,E1 13881.608,E2 13881.608} C_VEL
LIN {X 0,Y 297.521,Z 416.914,A -85,B 0,C 180,E1 13880.876,E2 13880.876} C_VEL
LIN {X 0,Y 294.059,Z 413.501,A -85,B 0,C 180,E1 13878.802,E2 13878.802} C_VEL
LIN {X 0,Y 292.541,Z 410.907,A -85,B 0,C 180,E1 13877.717,E2 13877.717} C_VEL
LIN {X 0,Y 289.097,Z 408.189,A -85,B 0,C 180,E1 13875.224,E2 13875.224} C_VEL
LIN {X 0,Y 287.058,Z 404.569,A -85,B 0,C 180,E1 13873.298,E2 13873.298} C_VEL
LIN {X 0,Y 282.928,Z 401.645,A -85,B 0,C 180,E1 13868.749,E2 13868.749} C_VEL
LIN {X 0,Y 281.176,Z 398.441,A -85,B 0,C 180,E1 13865.313,E2 13865.313} C_VEL
LIN {X 0,Y 280.1,Z 397.526,A -85,B 0,C 180,E1 13861.441,E2 13861.441} C_VEL
LIN {X 0,Y 280.651,Z 397.868,A -85,B 0,C 180,E1 13855.719,E2 13855.719} C_VEL
LIN {X 0,Y 281.547,Z 399.13,A -85,B 0,C 180,E1 13853.382,E2 13853.382} C_VEL
LIN {X 0,Y 284.116,Z 402.854,A -85,B 0,C 180,E1 13849.26,E2 13849.26} C_VEL
LIN {X 0,Y 287.288,Z 404.884,A -85,B 0,C 180,E1 13846.064,E2 13846.064} C_VEL
LIN {X 0,Y 289.572,Z 408.732,A -85,B 0,C 180,E1 13843.975,E2 13843.975} C_VEL
LIN {X 0,Y 292.852,Z 411.363,A -85,B 0,C 180,E1 13841.645,E2 13841.645} C_VEL
LIN {X 0,Y 295.254,Z 415.073,A -85,B 0,C 180,E1 13840.01,E2 13840.01} C_VEL
LIN {X 0,Y 298.048,Z 417.523,A -85,B 0,C 180,E1 13838.407,E2 13838.407} C_VEL
LIN {X 0,Y 301.073,Z 421.689,A -85,B 0,C 180,E1 13836.733,E2 13836.733} C_VEL
LIN {X 0,Y 302.947,Z 423.658,A -85,B 0,C 180,E1 13835.801,E2 13835.801} C_VEL
LIN {X 0,Y 306.545,Z 428.139,A -85,B 0,C 180,E1 13834.094,E2 13834.094} C_VEL
LIN {X 0,Y 308.828,Z 430.454,A -85,B 0,C 180,E1 13833.11,E2 13833.11} C_VEL
LIN {X 0,Y 313.205,Z 435.116,A -85,B 0,C 180,E1 13831.297,E2 13831.297} C_VEL
LIN {X 0,Y 316.031,Z 437.524,A -85,B 0,C 180,E1 13830.114,E2 13830.114} C_VEL
LIN {X 0,Y 320.341,Z 441.981,A -85,B 0,C 180,E1 13828.176,E2 13828.176} C_VEL
LIN {X 0,Y 324.181,Z 444.963,A -85,B 0,C 180,E1 13826.38,E2 13826.38} C_VEL
LIN {X 0,Y 328.267,Z 449.282,A -85,B 0,C 180,E1 13824.223,E2 13824.223} C_VEL
LIN {X 0,Y 331.549,Z 451.914,A -85,B 0,C 180,E1 13822.374,E2 13822.374} C_VEL
LIN {X 0,Y 334.898,Z 455.867,A -85,B 0,C 180,E1 13820.302,E2 13820.302} C_VEL
LIN {X 0,Y 338.805,Z 459.109,A -85,B 0,C 180,E1 13817.954,E2 13817.954} C_VEL
LIN {X 0,Y 342.814,Z 463.637,A -85,B 0,C 180,E1 13815.354,E2 13815.354} C_VEL
LIN {X 0,Y 345.978,Z 466.085,A -85,B 0,C 180,E1 13813.334,E2 13813.334} C_VEL
LIN {X 0,Y 349.582,Z 470.237,A -85,B 0,C 180,E1 13810.871,E2 13810.871} C_VEL
LIN {X 0,Y 353.381,Z 473.15,A -85,B 0,C 180,E1 13808.234,E2 13808.234} C_VEL
LIN {X 0,Y 356.943,Z 477.295,A -85,B 0,C 180,E1 13805.555,E2 13805.555} C_VEL
LIN {X 0,Y 360.362,Z 479.73,A -85,B 0,C 180,E1 13802.943,E2 13802.943} C_VEL
LIN {X 0,Y 361.428,Z 480.749,A -85,B 0,C 180,E1 13802.082,E2 13802.082} C_VEL
LIN {X 0,Y 364.243,Z 484.185,A -85,B 0,C 180,E1 13799.61,E2 13799.61} C_VEL
LIN {X 0,Y 367.361,Z 486.592,A -85,B 0,C 180,E1 13796.805,E2 13796.805} C_VEL
LIN {X 0,Y 369.363,Z 487.861,A -85,B 0,C 180,E1 13794.893,E2 13794.893} C_VEL
LIN {X 0,Y 371.729,Z 491.08,A -85,B 0,C 180,E1 13792.287,E2 13792.287} C_VEL
LIN {X 0,Y 374.451,Z 493.437,A -85,B 0,C 180,E1 13789.011,E2 13789.011} C_VEL
LIN {X 0,Y 376.905,Z 494.631,A -85,B 0,C 180,E1 13785.68,E2 13785.68} C_VEL
LIN {X 0,Y 378.051,Z 495.686,A -85,B 0,C 180,E1 13783.77,E2 13783.77} C_VEL
LIN {X 0,Y 379.54,Z 498.044,A -85,B 0,C 180,E1 13780.626,E2 13780.626} C_VEL
LIN {X 0,Y 380.693,Z 499.401,A -85,B 0,C 180,E1 13777.394,E2 13777.394} C_VEL
LIN {X 0,Y 381.514,Z 500.102,A -85,B 0,C 180,E1 13774.058,E2 13774.058} C_VEL
LIN {X 0,Y 381.838,Z 500.343,A -85,B 0,C 180,E1 13770.75,E2 13770.75} C_VEL
LIN {X 0,Y 381.716,Z 500.245,A -85,B 0,C 180,E1 13767.298,E2 13767.298} C_VEL
LIN {X 0,Y 381.103,Z 499.735,A -85,B 0,C 180,E1 13763.976,E2 13763.976} C_VEL
LIN {X 0,Y 380.012,Z 498.67,A -85,B 0,C 180,E1 13760.569,E2 13760.569} C_VEL
LIN {X 0,Y 378.711,Z 496.782,A -85,B 0,C 180,E1 13757.497,E2 13757.497} C_VEL
LIN {X 0,Y 377.308,Z 494.833,A -85,B 0,C 180,E1 13754.948,E2 13754.948} C_VEL
LIN {X 0,Y 374.837,Z 493.674,A -85,B 0,C 180,E1 13751.493,E2 13751.493} C_VEL
LIN {X 0,Y 372.154,Z 491.556,A -85,B 0,C 180,E1 13748.238,E2 13748.238} C_VEL
LIN {X 0,Y 369.699,Z 488.432,A -85,B 0,C 180,E1 13745.472,E2 13745.472} C_VEL
LIN {X 0,Y 368.749,Z 487.292,A -85,B 0,C 180,E1 13744.462,E2 13744.462} C_VEL
LIN {X 0,Y 365.582,Z 485.394,A -85,B 0,C 180,E1 13741.584,E2 13741.584} C_VEL
LIN {X 0,Y 362.376,Z 482.101,A -85,B 0,C 180,E1 13738.754,E2 13738.754} C_VEL
LIN {X 0,Y 360.662,Z 479.876,A -85,B 0,C 180,E1 13737.277,E2 13737.277} C_VEL
LIN {X 0,Y 357.12,Z 477.468,A -85,B 0,C 180,E1 13734.582,E2 13734.582} C_VEL
LIN {X 0,Y 353.468,Z 473.28,A -85,B 0,C 180,E1 13731.832,E2 13731.832} C_VEL
LIN {X 0,Y 351.756,Z 471.928,A -85,B 0,C 180,E1 13730.622,E2 13730.622} C_VEL
LIN {X 0,Y 348.007,Z 468.671,A -85,B 0,C 180,E1 13728.069,E2 13728.069} C_VEL
LIN {X 0,Y 345.199,Z 465.299,A -85,B 0,C 180,E1 13726.141,E2 13726.141} C_VEL
LIN {X 0,Y 341.373,Z 462.233,A -85,B 0,C 180,E1 13723.713,E2 13723.713} C_VEL
LIN {X 0,Y 337.907,Z 458.192,A -85,B 0,C 180,E1 13721.501,E2 13721.501} C_VEL
LIN {X 0,Y 333.729,Z 454.702,A -85,B 0,C 180,E1 13718.975,E2 13718.975} C_VEL
LIN {X 0,Y 330.801,Z 451.15,A -85,B 0,C 180,E1 13717.181,E2 13717.181} C_VEL
LIN {X 0,Y 326.622,Z 447.776,A -85,B 0,C 180,E1 13714.909,E2 13714.909} C_VEL
LIN {X 0,Y 323.074,Z 443.96,A -85,B 0,C 180,E1 13713.097,E2 13713.097} C_VEL
LIN {X 0,Y 318.698,Z 440.49,A -85,B 0,C 180,E1 13711.078,E2 13711.078} C_VEL
LIN {X 0,Y 314.63,Z 436.195,A -85,B 0,C 180,E1 13709.289,E2 13709.289} C_VEL
LIN {X 0,Y 310.122,Z 432.093,A -85,B 0,C 180,E1 13707.443,E2 13707.443} C_VEL
LIN {X 0,Y 307.543,Z 428.989,A -85,B 0,C 180,E1 13706.334,E2 13706.334} C_VEL
LIN {X 0,Y 303.643,Z 424.761,A -85,B 0,C 180,E1 13704.554,E2 13704.554} C_VEL
LIN {X 0,Y 302.153,Z 422.648,A -85,B 0,C 180,E1 13703.8,E2 13703.8} C_VEL
LIN {X 0,Y 298.738,Z 418.732,A -85,B 0,C 180,E1 13702.005,E2 13702.005} C_VEL
LIN {X 0,Y 297.487,Z 416.894,A -85,B 0,C 180,E1 13701.273,E2 13701.273} C_VEL
LIN {X 0,Y 294.162,Z 413.723,A -85,B 0,C 180,E1 13699.292,E2 13699.292} C_VEL
LIN {X 0,Y 292.512,Z 410.87,A -85,B 0,C 180,E1 13698.112,E2 13698.112} C_VEL
LIN {X 0,Y 289.099,Z 408.178,A -85,B 0,C 180,E1 13695.64,E2 13695.64} C_VEL
LIN {X 0,Y 286.931,Z 404.439,A -85,B 0,C 180,E1 13693.594,E2 13693.594} C_VEL
LIN {X 0,Y 283.053,Z 401.759,A -85,B 0,C 180,E1 13689.342,E2 13689.342} C_VEL
LIN {X 0,Y 281.01,Z 398.2,A -85,B 0,C 180,E1 13685.299,E2 13685.299} C_VEL
LIN {X 0,Y 280.018,Z 397.476,A -85,B 0,C 180,E1 13681.014,E2 13681.014} C_VEL
LIN {X 0,Y 280.796,Z 397.978,A -85,B 0,C 180,E1 13675.703,E2 13675.703} C_VEL
LIN {X 0,Y 281.741,Z 399.547,A -85,B 0,C 180,E1 13673.368,E2 13673.368} C_VEL
LIN {X 0,Y 284.301,Z 403.029,A -85,B 0,C 180,E1 13669.454,E2 13669.454} C_VEL
LIN {X 0,Y 287.318,Z 404.857,A -85,B 0,C 180,E1 13666.458,E2 13666.458} C_VEL
LIN {X 0,Y 289.24,Z 408.363,A -85,B 0,C 180,E1 13664.658,E2 13664.658} C_VEL
LIN {X 0,Y 292.871,Z 411.389,A -85,B 0,C 180,E1 13662.047,E2 13662.047} C_VEL
LIN {X 0,Y 295.445,Z 415.193,A -85,B 0,C 180,E1 13660.315,E2 13660.315} C_VEL
LIN {X 0,Y 297.941,Z 417.383,A -85,B 0,C 180,E1 13658.885,E2 13658.885} C_VEL
LIN {X 0,Y 300.319,Z 423.252,A -85,B 0,C 180,E1 13657.394,E2 13657.394} C_VEL
LIN {X 0,Y 304.819,Z 435.541,A -85,B 0,C 180,E1 13654.791,E2 13654.791} C_VEL
LIN {X 0,Y 306.916,Z 439.002,A -85,B 0,C 180,E1 13653.801,E2 13653.801} C_VEL
LIN {X 0,Y 309.903,Z 442.923,A -85,B 0,C 180,E1 13652.518,E2 13652.518} C_VEL
LIN {X 0,Y 312.884,Z 447.12,A -85,B 0,C 180,E1 13651.299,E2 13651.299} C_VEL
LIN {X 0,Y 319.501,Z 458.186,A -85,B 0,C 180,E1 13648.748,E2 13648.748} C_VEL
LIN {X 0,Y 326.969,Z 471.644,A -85,B 0,C 180,E1 13646.15,E2 13646.15} C_VEL
LIN {X 0,Y 334.964,Z 487.756,A -85,B 0,C 180,E1 13643.605,E2 13643.605} C_VEL
LIN {X 0,Y 335.462,Z 489.275,A -85,B 0,C 180,E1 13643.437,E2 13643.437} C_VEL
LIN {X 0,Y 325.994,Z 644.139,A -85,B 0,C 180,E1 13640.129,E2 13640.129} C_VEL
LIN {X 0,Y 323.512,Z 665.429,A -85,B 0,C 180,E1 13639.471,E2 13639.471} C_VEL
LIN {X 0,Y 320.314,Z 683.95,A -85,B 0,C 180,E1 13638.651,E2 13638.651} C_VEL
LIN {X 0,Y 316.894,Z 700.183,A -85,B 0,C 180,E1 13637.72,E2 13637.72} C_VEL
LIN {X 0,Y 312.252,Z 719.01,A -85,B 0,C 180,E1 13636.357,E2 13636.357} C_VEL
LIN {X 0,Y 307.015,Z 736.759,A -85,B 0,C 180,E1 13634.703,E2 13634.703} C_VEL
LIN {X 0,Y 302.313,Z 751.186,A -85,B 0,C 180,E1 13633.075,E2 13633.075} C_VEL
LIN {X 0,Y 296.526,Z 767.57,A -85,B 0,C 180,E1 13630.854,E2 13630.854} C_VEL
LIN {X 0,Y 290.597,Z 782.885,A -85,B 0,C 180,E1 13628.266,E2 13628.266} C_VEL
LIN {X 0,Y 285.623,Z 795.205,A -85,B 0,C 180,E1 13625.774,E2 13625.774} C_VEL
LIN {X 0,Y 280.236,Z 808.354,A -85,B 0,C 180,E1 13622.598,E2 13622.598} C_VEL
LIN {X 0,Y 275.395,Z 819.946,A -85,B 0,C 180,E1 13619.11,E2 13619.11} C_VEL
LIN {X 0,Y 271.901,Z 828.701,A -85,B 0,C 180,E1 13615.95,E2 13615.95} C_VEL
LIN {X 0,Y 268.608,Z 837.695,A -85,B 0,C 180,E1 13612.034,E2 13612.034} C_VEL
LIN {X 0,Y 266.138,Z 845.352,A -85,B 0,C 180,E1 13607.716,E2 13607.716} C_VEL
LIN {X 0,Y 264.843,Z 850.53,A -85,B 0,C 180,E1 13603.982,E2 13603.982} C_VEL
LIN {X 0,Y 264.145,Z 854.886,A -85,B 0,C 180,E1 13599.807,E2 13599.807} C_VEL
LIN {X 0,Y 263.962,Z 857.692,A -85,B 0,C 180,E1 13595.434,E2 13595.434} C_VEL
LIN {X 0,Y 263.979,Z 858.786,A -85,B 0,C 180,E1 13591.953,E2 13591.953} C_VEL
LIN {X 0,Y 263.988,Z 858.876,A -85,B 0,C 180,E1 13588.698,E2 13588.698} C_VEL
LIN {X 0,Y 263.96,Z 857.961,A -85,B 0,C 180,E1 13585.22,E2 13585.22} C_VEL
LIN {X 0,Y 264.032,Z 856.005,A -85,B 0,C 180,E1 13581.727,E2 13581.727} C_VEL
LIN {X 0,Y 264.504,Z 852.36,A -85,B 0,C 180,E1 13577.557,E2 13577.557} C_VEL
LIN {X 0,Y 265.772,Z 846.696,A -85,B 0,C 180,E1 13573.162,E2 13573.162} C_VEL
LIN {X 0,Y 267.632,Z 840.477,A -85,B 0,C 180,E1 13569.441,E2 13569.441} C_VEL
LIN {X 0,Y 270.713,Z 831.916,A -85,B 0,C 180,E1 13565.323,E2 13565.323} C_VEL
LIN {X 0,Y 274.639,Z 821.811,A -85,B 0,C 180,E1 13561.516,E2 13561.516} C_VEL
LIN {X 0,Y 278.71,Z 811.894,A -85,B 0,C 180,E1 13558.416,E2 13558.416} C_VEL
LIN {X 0,Y 284.001,Z 799.281,A -85,B 0,C 180,E1 13555.125,E2 13555.125} C_VEL
LIN {X 0,Y 289.598,Z 785.389,A -85,B 0,C 180,E1 13552.207,E2 13552.207} C_VEL
LIN {X 0,Y 294.552,Z 772.679,A -85,B 0,C 180,E1 13549.966,E2 13549.966} C_VEL
LIN {X 0,Y 300.343,Z 757.048,A -85,B 0,C 180,E1 13547.658,E2 13547.658} C_VEL
LIN {X 0,Y 305.999,Z 739.987,A -85,B 0,C 180,E1 13545.635,E2 13545.635} C_VEL
LIN {X 0,Y 310.639,Z 724.553,A -85,B 0,C 180,E1 13544.131,E2 13544.131} C_VEL
LIN {X 0,Y 315.516,Z 706.283,A -85,B 0,C 180,E1 13542.678,E2 13542.678} C_VEL
LIN {X 0,Y 319.715,Z 687.075,A -85,B 0,C 180,E1 13541.512,E2 13541.512} C_VEL
LIN {X 0,Y 322.736,Z 670.198,A -85,B 0,C 180,E1 13540.723,E2 13540.723} C_VEL
LIN {X 0,Y 325.366,Z 651.023,A -85,B 0,C 180,E1 13540.053,E2 13540.053} C_VEL
LIN {X 0,Y 327.473,Z 622.274,A -85,B 0,C 180,E1 13539.374,E2 13539.374} C_VEL
LIN {X 0,Y 335.392,Z 488.717,A -85,B 0,C 180,E1 13536.527,E2 13536.527} C_VEL
LIN {X 0,Y 327.731,Z 473.123,A -85,B 0,C 180,E1 13534.103,E2 13534.103} C_VEL
LIN {X 0,Y 320.61,Z 460.125,A -85,B 0,C 180,E1 13531.655,E2 13531.655} C_VEL
LIN {X 0,Y 314.867,Z 450.308,A -85,B 0,C 180,E1 13529.492,E2 13529.492} C_VEL
LIN {X 0,Y 311.234,Z 444.689,A -85,B 0,C 180,E1 13528.031,E2 13528.031} C_VEL
LIN {X 0,Y 307.314,Z 439.494,A -85,B 0,C 180,E1 13526.373,E2 13526.373} C_VEL
LIN {X 0,Y 303.9,Z 434.952,A -85,B 0,C 180,E1 13524.809,E2 13524.809} C_VEL
LIN {X 0,Y 299.982,Z 429.943,A -85,B 0,C 180,E1 13522.856,E2 13522.856} C_VEL
LIN {X 0,Y 296.511,Z 425.716,A -85,B 0,C 180,E1 13520.95,E2 13520.95} C_VEL
LIN {X 0,Y 295.433,Z 424.266,A -85,B 0,C 180,E1 13520.305,E2 13520.305} C_VEL
LIN {X 0,Y 292.037,Z 420.549,A -85,B 0,C 180,E1 13518.161,E2 13518.161} C_VEL
LIN {X 0,Y 290.74,Z 418.505,A -85,B 0,C 180,E1 13517.21,E2 13517.21} C_VEL
LIN {X 0,Y 287.241,Z 415.314,A -85,B 0,C 180,E1 13514.522,E2 13514.522} C_VEL
LIN {X 0,Y 285.674,Z 412.286,A -85,B 0,C 180,E1 13512.952,E2 13512.952} C_VEL
LIN {X 0,Y 281.949,Z 409.714,A -85,B 0,C 180,E1 13508.779,E2 13508.779} C_VEL
LIN {X 0,Y 280.118,Z 406.319,A -85,B 0,C 180,E1 13505.128,E2 13505.128} C_VEL
LIN {X 0,Y 279.125,Z 405.467,A -85,B 0,C 180,E1 13501.446,E2 13501.446} C_VEL
LIN {X 0,Y 279.677,Z 405.823,A -85,B 0,C 180,E1 13495.704,E2 13495.704} C_VEL
LIN {X 0,Y 280.516,Z 407.134,A -85,B 0,C 180,E1 13493.46,E2 13493.46} C_VEL
LIN {X 0,Y 283.15,Z 410.866,A -85,B 0,C 180,E1 13489.223,E2 13489.223} C_VEL
LIN {X 0,Y 285.842,Z 412.593,A -85,B 0,C 180,E1 13486.456,E2 13486.456} C_VEL
LIN {X 0,Y 288.125,Z 416.421,A -85,B 0,C 180,E1 13484.306,E2 13484.306} C_VEL
LIN {X 0,Y 291.177,Z 419.028,A -85,B 0,C 180,E1 13482.06,E2 13482.06} C_VEL
LIN {X 0,Y 293.842,Z 422.927,A -85,B 0,C 180,E1 13480.221,E2 13480.221} C_VEL
LIN {X 0,Y 296.19,Z 425.094,A -85,B 0,C 180,E1 13478.836,E2 13478.836} C_VEL
LIN {X 0,Y 299.423,Z 429.406,A -85,B 0,C 180,E1 13477.013,E2 13477.013} C_VEL
LIN {X 0,Y 300.988,Z 431.238,A -85,B 0,C 180,E1 13476.207,E2 13476.207} C_VEL
LIN {X 0,Y 304.828,Z 435.863,A -85,B 0,C 180,E1 13474.355,E2 13474.355} C_VEL
LIN {X 0,Y 306.871,Z 438.125,A -85,B 0,C 180,E1 13473.447,E2 13473.447} C_VEL
LIN {X 0,Y 311.455,Z 442.835,A -85,B 0,C 180,E1 13471.54,E2 13471.54} C_VEL
LIN {X 0,Y 314.099,Z 445.137,A -85,B 0,C 180,E1 13470.447,E2 13470.447} C_VEL
LIN {X 0,Y 318.693,Z 449.71,A -85,B 0,C 180,E1 13468.415,E2 13468.415} C_VEL
LIN {X 0,Y 322.445,Z 452.659,A -85,B 0,C 180,E1 13466.67,E2 13466.67} C_VEL
LIN {X 0,Y 326.67,Z 456.957,A -85,B 0,C 180,E1 13464.502,E2 13464.502} C_VEL
LIN {X 0,Y 330.005,Z 459.644,A -85,B 0,C 180,E1 13462.66,E2 13462.66} C_VEL
LIN {X 0,Y 333.605,Z 463.746,A -85,B 0,C 180,E1 13460.453,E2 13460.453} C_VEL
LIN {X 0,Y 337.213,Z 466.717,A -85,B 0,C 180,E1 13458.281,E2 13458.281} C_VEL
LIN {X 0,Y 341.419,Z 471.384,A -85,B 0,C 180,E1 13455.594,E2 13455.594} C_VEL
LIN {X 0,Y 344.577,Z 473.864,A -85,B 0,C 180,E1 13453.577,E2 13453.577} C_VEL
LIN {X 0,Y 348.179,Z 477.97,A -85,B 0,C 180,E1 13451.117,E2 13451.117} C_VEL
LIN {X 0,Y 352.108,Z 481.032,A -85,B 0,C 180,E1 13448.412,E2 13448.412} C_VEL
LIN {X 0,Y 355.747,Z 485.164,A -85,B 0,C 180,E1 13445.7,E2 13445.7} C_VEL
LIN {X 0,Y 359.201,Z 487.611,A -85,B 0,C 180,E1 13443.063,E2 13443.063} C_VEL
LIN {X 0,Y 360.396,Z 488.901,A -85,B 0,C 180,E1 13442.088,E2 13442.088} C_VEL
LIN {X 0,Y 363.359,Z 492.316,A -85,B 0,C 180,E1 13439.508,E2 13439.508} C_VEL
LIN {X 0,Y 366.419,Z 494.574,A -85,B 0,C 180,E1 13436.758,E2 13436.758} C_VEL
LIN {X 0,Y 368.198,Z 495.729,A -85,B 0,C 180,E1 13435.063,E2 13435.063} C_VEL
LIN {X 0,Y 370.503,Z 498.846,A -85,B 0,C 180,E1 13432.532,E2 13432.532} C_VEL
LIN {X 0,Y 373.149,Z 501.18,A -85,B 0,C 180,E1 13429.405,E2 13429.405} C_VEL
LIN {X 0,Y 375.688,Z 502.48,A -85,B 0,C 180,E1 13426.068,E2 13426.068} C_VEL
LIN {X 0,Y 376.983,Z 503.534,A -85,B 0,C 180,E1 13423.942,E2 13423.942} C_VEL
LIN {X 0,Y 378.492,Z 505.916,A -85,B 0,C 180,E1 13420.81,E2 13420.81} C_VEL
LIN {X 0,Y 379.67,Z 507.286,A -85,B 0,C 180,E1 13417.566,E2 13417.566} C_VEL
LIN {X 0,Y 380.516,Z 508.021,A -85,B 0,C 180,E1 13414.219,E2 13414.219} C_VEL
LIN {X 0,Y 380.86,Z 508.269,A -85,B 0,C 180,E1 13410.903,E2 13410.903} C_VEL
LIN {X 0,Y 380.752,Z 508.204,A -85,B 0,C 180,E1 13407.441,E2 13407.441} C_VEL
LIN {X 0,Y 380.154,Z 507.703,A -85,B 0,C 180,E1 13404.113,E2 13404.113} C_VEL
LIN {X 0,Y 379.095,Z 506.708,A -85,B 0,C 180,E1 13400.742,E2 13400.742} C_VEL
LIN {X 0,Y 377.715,Z 504.747,A -85,B 0,C 180,E1 13397.464,E2 13397.464} C_VEL
LIN {X 0,Y 376.3,Z 502.765,A -85,B 0,C 180,E1 13394.907,E2 13394.907} C_VEL
LIN {X 0,Y 373.814,Z 501.601,A -85,B 0,C 180,E1 13391.441,E2 13391.441} C_VEL
LIN {X 0,Y 371.109,Z 499.491,A -85,B 0,C 180,E1 13388.174,E2 13388.174} C_VEL
LIN {X 0,Y 368.531,Z 496.291,A -85,B 0,C 180,E1 13385.304,E2 13385.304} C_VEL
LIN {X 0,Y 367.685,Z 495.205,A -85,B 0,C 180,E1 13384.383,E2 13384.383} C_VEL
LIN {X 0,Y 364.374,Z 493.211,A -85,B 0,C 180,E1 13381.392,E2 13381.392} C_VEL
LIN {X 0,Y 361.071,Z 489.84,A -85,B 0,C 180,E1 13378.508,E2 13378.508} C_VEL
LIN {X 0,Y 359.455,Z 487.736,A -85,B 0,C 180,E1 13377.125,E2 13377.125} C_VEL
LIN {X 0,Y 355.932,Z 485.345,A -85,B 0,C 180,E1 13374.446,E2 13374.446} C_VEL
LIN {X 0,Y 352.243,Z 481.227,A -85,B 0,C 180,E1 13371.691,E2 13371.691} C_VEL
LIN {X 0,Y 350.974,Z 480.048,A -85,B 0,C 180,E1 13370.771,E2 13370.771} C_VEL
LIN {X 0,Y 347.049,Z 476.879,A -85,B 0,C 180,E1 13368.122,E2 13368.122} C_VEL
LIN {X 0,Y 343.81,Z 473.067,A -85,B 0,C 180,E1 13365.901,E2 13365.901} C_VEL
LIN {X 0,Y 339.947,Z 469.986,A -85,B 0,C 180,E1 13363.477,E2 13363.477} C_VEL
LIN {X 0,Y 336.46,Z 465.936,A -85,B 0,C 180,E1 13361.252,E2 13361.252} C_VEL
LIN {X 0,Y 331.991,Z 462.142,A -85,B 0,C 180,E1 13358.554,E2 13358.554} C_VEL
LIN {X 0,Y 329.178,Z 458.797,A -85,B 0,C 180,E1 13356.85,E2 13356.85} C_VEL
LIN {X 0,Y 324.905,Z 455.367,A -85,B 0,C 180,E1 13354.583,E2 13354.583} C_VEL
LIN {X 0,Y 321.298,Z 451.572,A -85,B 0,C 180,E1 13352.772,E2 13352.772} C_VEL
LIN {X 0,Y 316.619,Z 447.85,A -85,B 0,C 180,E1 13350.653,E2 13350.653} C_VEL
LIN {X 0,Y 312.518,Z 443.613,A -85,B 0,C 180,E1 13348.877,E2 13348.877} C_VEL
LIN {X 0,Y 307.754,Z 439.235,A -85,B 0,C 180,E1 13346.939,E2 13346.939} C_VEL
LIN {X 0,Y 305.221,Z 436.206,A -85,B 0,C 180,E1 13345.818,E2 13345.818} C_VEL
LIN {X 0,Y 301.243,Z 431.644,A -85,B 0,C 180,E1 13343.928,E2 13343.928} C_VEL
LIN {X 0,Y 299.775,Z 429.735,A -85,B 0,C 180,E1 13343.166,E2 13343.166} C_VEL
LIN {X 0,Y 296.338,Z 425.362,A -85,B 0,C 180,E1 13341.256,E2 13341.256} C_VEL
LIN {X 0,Y 295.24,Z 424.137,A -85,B 0,C 180,E1 13340.612,E2 13340.612} C_VEL
LIN {X 0,Y 292.071,Z 420.671,A -85,B 0,C 180,E1 13338.606,E2 13338.606} C_VEL
LIN {X 0,Y 290.719,Z 418.43,A -85,B 0,C 180,E1 13337.607,E2 13337.607} C_VEL
LIN {X 0,Y 287.439,Z 415.574,A -85,B 0,C 180,E1 13335.113,E2 13335.113} C_VEL
LIN {X 0,Y 285.65,Z 412.283,A -85,B 0,C 180,E1 13333.347,E2 13333.347} C_VEL
LIN {X 0,Y 281.806,Z 409.482,A -85,B 0,C 180,E1 13328.972,E2 13328.972} C_VEL
LIN {X 0,Y 279.958,Z 406.087,A -85,B 0,C 180,E1 13325.113,E2 13325.113} C_VEL
LIN {X 0,Y 279.03,Z 405.418,A -85,B 0,C 180,E1 13320.812,E2 13320.812} C_VEL
LIN {X 0,Y 279.822,Z 405.934,A -85,B 0,C 180,E1 13315.688,E2 13315.688} C_VEL
LIN {X 0,Y 280.656,Z 407.473,A -85,B 0,C 180,E1 13313.548,E2 13313.548} C_VEL
LIN {X 0,Y 283.334,Z 411.036,A -85,B 0,C 180,E1 13309.418,E2 13309.418} C_VEL
LIN {X 0,Y 285.866,Z 412.599,A -85,B 0,C 180,E1 13306.851,E2 13306.851} C_VEL
LIN {X 0,Y 287.914,Z 416.187,A -85,B 0,C 180,E1 13304.895,E2 13304.895} C_VEL
LIN {X 0,Y 291.205,Z 419.051,A -85,B 0,C 180,E1 13302.457,E2 13302.457} C_VEL
LIN {X 0,Y 294.029,Z 423.044,A -85,B 0,C 180,E1 13300.526,E2 13300.526} C_VEL
LIN {X 0,Y 296.212,Z 425.196,A -85,B 0,C 180,E1 13299.234,E2 13299.234} C_VEL
LIN {X 0,Y 299.452,Z 429.461,A -85,B 0,C 180,E1 13297.412,E2 13297.412} C_VEL
LIN {X 0,Y 301.112,Z 431.346,A -85,B 0,C 180,E1 13296.562,E2 13296.562} C_VEL
LIN {X 0,Y 305.585,Z 437.162,A -85,B 0,C 180,E1 13294.405,E2 13294.405} C_VEL
LIN {X 0,Y 306.916,Z 439.002,A -85,B 0,C 180,E1 13293.801,E2 13293.801} C_VEL
LIN {X 0,Y 308.997,Z 442.704,A -85,B 0,C 180,E1 13292.85,E2 13292.85} C_VEL
LIN {X 0,Y 311.434,Z 449.979,A -85,B 0,C 180,E1 13291.65,E2 13291.65} C_VEL
LIN {X 0,Y 314.841,Z 461.255,A -85,B 0,C 180,E1 13290.026,E2 13290.026} C_VEL
LIN {X 0,Y 316.214,Z 464.287,A -85,B 0,C 180,E1 13289.469,E2 13289.469} C_VEL
LIN {X 0,Y 323.556,Z 477.868,A -85,B 0,C 180,E1 13286.808,E2 13286.808} C_VEL
LIN {X 0,Y 330.538,Z 492.224,A -85,B 0,C 180,E1 13284.488,E2 13284.488} C_VEL
LIN {X 0,Y 320.91,Z 643.884,A -85,B 0,C 180,E1 13281.23,E2 13281.23} C_VEL
LIN {X 0,Y 318.371,Z 665.077,A -85,B 0,C 180,E1 13280.575,E2 13280.575} C_VEL
LIN {X 0,Y 315.055,Z 683.713,A -85,B 0,C 180,E1 13279.75,E2 13279.75} C_VEL
LIN {X 0,Y 311.527,Z 699.944,A -85,B 0,C 180,E1 13278.818,E2 13278.818} C_VEL
LIN {X 0,Y 306.727,Z 718.771,A -85,B 0,C 180,E1 13277.45,E2 13277.45} C_VEL
LIN {X 0,Y 301.308,Z 736.519,A -85,B 0,C 180,E1 13275.787,E2 13275.787} C_VEL
LIN {X 0,Y 296.428,Z 750.946,A -85,B 0,C 180,E1 13274.148,E2 13274.148} C_VEL
LIN {X 0,Y 290.407,Z 767.329,A -85,B 0,C 180,E1 13271.906,E2 13271.906} C_VEL
LIN {X 0,Y 284.19,Z 782.708,A -85,B 0,C 180,E1 13269.275,E2 13269.275} C_VEL
LIN {X 0,Y 279.015,Z 794.963,A -85,B 0,C 180,E1 13266.758,E2 13266.758} C_VEL
LIN {X 0,Y 273.353,Z 808.111,A -85,B 0,C 180,E1 13263.525,E2 13263.525} C_VEL
LIN {X 0,Y 268.243,Z 819.703,A -85,B 0,C 180,E1 13259.964,E2 13259.964} C_VEL
LIN {X 0,Y 264.533,Z 828.458,A -85,B 0,C 180,E1 13256.729,E2 13256.729} C_VEL
LIN {X 0,Y 261.051,Z 837.352,A -85,B 0,C 180,E1 13252.757,E2 13252.757} C_VEL
LIN {X 0,Y 258.463,Z 844.773,A -85,B 0,C 180,E1 13248.494,E2 13248.494} C_VEL
LIN {X 0,Y 257.008,Z 850.017,A -85,B 0,C 180,E1 13244.647,E2 13244.647} C_VEL
LIN {X 0,Y 256.245,Z 854.016,A -85,B 0,C 180,E1 13240.795,E2 13240.795} C_VEL
LIN {X 0,Y 255.966,Z 857.274,A -85,B 0,C 180,E1 13236.054,E2 13236.054} C_VEL
LIN {X 0,Y 255.978,Z 858.52,A -85,B 0,C 180,E1 13232.238,E2 13232.238} C_VEL
LIN {X 0,Y 255.993,Z 858.669,A -85,B 0,C 180,E1 13228.881,E2 13228.881} C_VEL
LIN {X 0,Y 255.961,Z 857.813,A -85,B 0,C 180,E1 13225.295,E2 13225.295} C_VEL
LIN {X 0,Y 256.033,Z 855.916,A -85,B 0,C 180,E1 13221.692,E2 13221.692} C_VEL
LIN {X 0,Y 256.447,Z 852.752,A -85,B 0,C 180,E1 13217.846,E2 13217.846} C_VEL
LIN {X 0,Y 257.777,Z 847.127,A -85,B 0,C 180,E1 13213.088,E2 13213.088} C_VEL
LIN {X 0,Y 259.689,Z 841.039,A -85,B 0,C 180,E1 13209.255,E2 13209.255} C_VEL
LIN {X 0,Y 262.297,Z 834.004,A -85,B 0,C 180,E1 13205.665,E2 13205.665} C_VEL
LIN {X 0,Y 266.427,Z 824.054,A -85,B 0,C 180,E1 13201.537,E2 13201.537} C_VEL
LIN {X 0,Y 271.128,Z 813.06,A -85,B 0,C 180,E1 13197.925,E2 13197.925} C_VEL
LIN {X 0,Y 275.723,Z 802.56,A -85,B 0,C 180,E1 13195.044,E2 13195.044} C_VEL
LIN {X 0,Y 281.756,Z 788.653,A -85,B 0,C 180,E1 13191.87,E2 13191.87} C_VEL
LIN {X 0,Y 287.68,Z 774.123,A -85,B 0,C 180,E1 13189.202,E2 13189.202} C_VEL
LIN {X 0,Y 293,Z 760.383,A -85,B 0,C 180,E1 13187.096,E2 13187.096} C_VEL
LIN {X 0,Y 299.223,Z 742.977,A -85,B 0,C 180,E1 13184.897,E2 13184.897} C_VEL
LIN {X 0,Y 304.514,Z 726.157,A -85,B 0,C 180,E1 13183.205,E2 13183.205} C_VEL
LIN {X 0,Y 308.949,Z 710.298,A -85,B 0,C 180,E1 13181.898,E2 13181.898} C_VEL
LIN {X 0,Y 313.588,Z 691.148,A -85,B 0,C 180,E1 13180.639,E2 13180.639} C_VEL
LIN {X 0,Y 317.263,Z 671.715,A -85,B 0,C 180,E1 13179.696,E2 13179.696} C_VEL
LIN {X 0,Y 319.788,Z 654.473,A -85,B 0,C 180,E1 13179.072,E2 13179.072} C_VEL
LIN {X 0,Y 321.797,Z 632.615,A -85,B 0,C 180,E1 13178.498,E2 13178.498} C_VEL
LIN {X 0,Y 330.418,Z 491.972,A -85,B 0,C 180,E1 13175.474,E2 13175.474} C_VEL
LIN {X 0,Y 322.753,Z 476.369,A -85,B 0,C 180,E1 13172.916,E2 13172.916} C_VEL
LIN {X 0,Y 314.886,Z 461.835,A -85,B 0,C 180,E1 13170.014,E2 13170.014} C_VEL
LIN {X 0,Y 308.714,Z 451.702,A -85,B 0,C 180,E1 13167.493,E2 13167.493} C_VEL
LIN {X 0,Y 304.4,Z 445.899,A -85,B 0,C 180,E1 13165.598,E2 13165.598} C_VEL
LIN {X 0,Y 301.451,Z 441.909,A -85,B 0,C 180,E1 13164.189,E2 13164.189} C_VEL
LIN {X 0,Y 297.807,Z 437.169,A -85,B 0,C 180,E1 13162.303,E2 13162.303} C_VEL
LIN {X 0,Y 294.298,Z 432.602,A -85,B 0,C 180,E1 13160.283,E2 13160.283} C_VEL
LIN {X 0,Y 289.989,Z 427.481,A -85,B 0,C 180,E1 13157.463,E2 13157.463} C_VEL
LIN {X 0,Y 289.24,Z 426.227,A -85,B 0,C 180,E1 13156.888,E2 13156.888} C_VEL
LIN {X 0,Y 285.822,Z 423.012,A -85,B 0,C 180,E1 13154.182,E2 13154.182} C_VEL
LIN {X 0,Y 284.294,Z 420.06,A -85,B 0,C 180,E1 13152.603,E2 13152.603} C_VEL
LIN {X 0,Y 280.707,Z 417.424,A -85,B 0,C 180,E1 13148.406,E2 13148.406} C_VEL
LIN {X 0,Y 278.989,Z 414.083,A -85,B 0,C 180,E1 13144.737,E2 13144.737} C_VEL
LIN {X 0,Y 278.069,Z 413.363,A -85,B 0,C 180,E1 13140.627,E2 13140.627} C_VEL
LIN {X 0,Y 278.769,Z 413.839,A -85,B 0,C 180,E1 13135.484,E2 13135.484} C_VEL
LIN {X 0,Y 279.572,Z 415.326,A -85,B 0,C 180,E1 13133.335,E2 13133.335} C_VEL
LIN {X 0,Y 282.184,Z 418.873,A -85,B 0,C 180,E1 13129.186,E2 13129.186} C_VEL
LIN {X 0,Y 284.455,Z 420.391,A -85,B 0,C 180,E1 13126.803,E2 13126.803} C_VEL
LIN {X 0,Y 286.803,Z 424.238,A -85,B 0,C 180,E1 13124.542,E2 13124.542} C_VEL
LIN {X 0,Y 289.47,Z 426.549,A -85,B 0,C 180,E1 13122.522,E2 13122.522} C_VEL
LIN {X 0,Y 292.287,Z 430.623,A -85,B 0,C 180,E1 13120.527,E2 13120.527} C_VEL
LIN {X 0,Y 294.351,Z 432.637,A -85,B 0,C 180,E1 13119.271,E2 13119.271} C_VEL
LIN {X 0,Y 297.781,Z 437.118,A -85,B 0,C 180,E1 13117.297,E2 13117.297} C_VEL
LIN {X 0,Y 302.733,Z 443.233,A -85,B 0,C 180,E1 13114.793,E2 13114.793} C_VEL
LIN {X 0,Y 305.216,Z 446.138,A -85,B 0,C 180,E1 13113.659,E2 13113.659} C_VEL
LIN {X 0,Y 310.13,Z 450.863,A -85,B 0,C 180,E1 13111.617,E2 13111.617} C_VEL
LIN {X 0,Y 312.962,Z 453.64,A -85,B 0,C 180,E1 13110.434,E2 13110.434} C_VEL
LIN {X 0,Y 317.802,Z 458.021,A -85,B 0,C 180,E1 13108.316,E2 13108.316} C_VEL
LIN {X 0,Y 320.6,Z 460.203,A -85,B 0,C 180,E1 13107.025,E2 13107.025} C_VEL
LIN {X 0,Y 324.865,Z 464.478,A -85,B 0,C 180,E1 13104.875,E2 13104.875} C_VEL
LIN {X 0,Y 328.456,Z 467.363,A -85,B 0,C 180,E1 13102.947,E2 13102.947} C_VEL
LIN {X 0,Y 332.213,Z 471.532,A -85,B 0,C 180,E1 13100.666,E2 13100.666} C_VEL
LIN {X 0,Y 335.774,Z 474.516,A -85,B 0,C 180,E1 13098.519,E2 13098.519} C_VEL
LIN {X 0,Y 340.016,Z 479.13,A -85,B 0,C 180,E1 13095.833,E2 13095.833} C_VEL
LIN {X 0,Y 343.128,Z 481.561,A -85,B 0,C 180,E1 13093.861,E2 13093.861} C_VEL
LIN {X 0,Y 346.965,Z 485.868,A -85,B 0,C 180,E1 13091.24,E2 13091.24} C_VEL
LIN {X 0,Y 350.798,Z 488.853,A -85,B 0,C 180,E1 13088.622,E2 13088.622} C_VEL
LIN {X 0,Y 354.538,Z 493.033,A -85,B 0,C 180,E1 13085.844,E2 13085.844} C_VEL
LIN {X 0,Y 358.111,Z 495.527,A -85,B 0,C 180,E1 13083.131,E2 13083.131} C_VEL
LIN {X 0,Y 361.77,Z 499.786,A -85,B 0,C 180,E1 13080.015,E2 13080.015} C_VEL
LIN {X 0,Y 365.133,Z 502.374,A -85,B 0,C 180,E1 13077.036,E2 13077.036} C_VEL
LIN {X 0,Y 367.037,Z 503.595,A -85,B 0,C 180,E1 13075.234,E2 13075.234} C_VEL
LIN {X 0,Y 369.442,Z 506.784,A -85,B 0,C 180,E1 13072.6,E2 13072.6} C_VEL
LIN {X 0,Y 372.125,Z 509.111,A -85,B 0,C 180,E1 13069.454,E2 13069.454} C_VEL
LIN {X 0,Y 374.675,Z 510.411,A -85,B 0,C 180,E1 13066.113,E2 13066.113} C_VEL
LIN {X 0,Y 375.968,Z 511.482,A -85,B 0,C 180,E1 13064.005,E2 13064.005} C_VEL
LIN {X 0,Y 377.5,Z 513.857,A -85,B 0,C 180,E1 13060.839,E2 13060.839} C_VEL
LIN {X 0,Y 378.687,Z 515.229,A -85,B 0,C 180,E1 13057.586,E2 13057.586} C_VEL
LIN {X 0,Y 379.52,Z 515.94,A -85,B 0,C 180,E1 13054.382,E2 13054.382} C_VEL
LIN {X 0,Y 379.879,Z 516.199,A -85,B 0,C 180,E1 13051.056,E2 13051.056} C_VEL
LIN {X 0,Y 379.805,Z 516.179,A -85,B 0,C 180,E1 13047.737,E2 13047.737} C_VEL
LIN {X 0,Y 379.24,Z 515.713,A -85,B 0,C 180,E1 13044.402,E2 13044.402} C_VEL
LIN {X 0,Y 378.166,Z 514.717,A -85,B 0,C 180,E1 13040.872,E2 13040.872} C_VEL
LIN {X 0,Y 376.781,Z 512.837,A -85,B 0,C 180,E1 13037.588,E2 13037.588} C_VEL
LIN {X 0,Y 375.291,Z 510.698,A -85,B 0,C 180,E1 13034.866,E2 13034.866} C_VEL
LIN {X 0,Y 372.922,Z 509.59,A -85,B 0,C 180,E1 13031.557,E2 13031.557} C_VEL
LIN {X 0,Y 370.213,Z 507.57,A -85,B 0,C 180,E1 13028.285,E2 13028.285} C_VEL
LIN {X 0,Y 367.516,Z 504.375,A -85,B 0,C 180,E1 13025.298,E2 13025.298} C_VEL
LIN {X 0,Y 366.473,Z 503.051,A -85,B 0,C 180,E1 13024.18,E2 13024.18} C_VEL
LIN {X 0,Y 363.165,Z 501.029,A -85,B 0,C 180,E1 13021.198,E2 13021.198} C_VEL
LIN {X 0,Y 359.843,Z 497.67,A -85,B 0,C 180,E1 13018.322,E2 13018.322} C_VEL
LIN {X 0,Y 358.044,Z 495.492,A -85,B 0,C 180,E1 13016.816,E2 13016.816} C_VEL
LIN {X 0,Y 354.391,Z 492.902,A -85,B 0,C 180,E1 13014.051,E2 13014.051} C_VEL
LIN {X 0,Y 350.654,Z 488.652,A -85,B 0,C 180,E1 13011.266,E2 13011.266} C_VEL
LIN {X 0,Y 346.03,Z 484.997,A -85,B 0,C 180,E1 13008.129,E2 13008.129} C_VEL
LIN {X 0,Y 342.408,Z 480.832,A -85,B 0,C 180,E1 13005.663,E2 13005.663} C_VEL
LIN {X 0,Y 338.524,Z 477.738,A -85,B 0,C 180,E1 13003.24,E2 13003.24} C_VEL
LIN {X 0,Y 334.757,Z 473.505,A -85,B 0,C 180,E1 13000.839,E2 13000.839} C_VEL
LIN {X 0,Y 330.085,Z 469.412,A -85,B 0,C 180,E1 12998.044,E2 12998.044} C_VEL
LIN {X 0,Y 327.523,Z 466.437,A -85,B 0,C 180,E1 12996.521,E2 12996.521} C_VEL
LIN {X 0,Y 323.02,Z 462.792,A -85,B 0,C 180,E1 12994.169,E2 12994.169} C_VEL
LIN {X 0,Y 319.34,Z 459.063,A -85,B 0,C 180,E1 12992.359,E2 12992.359} C_VEL
LIN {X 0,Y 314.338,Z 455.049,A -85,B 0,C 180,E1 12990.159,E2 12990.159} C_VEL
LIN {X 0,Y 310.341,Z 451.015,A -85,B 0,C 180,E1 12988.467,E2 12988.467} C_VEL
LIN {X 0,Y 305.313,Z 446.259,A -85,B 0,C 180,E1 12986.384,E2 12986.384} C_VEL
LIN {X 0,Y 302.925,Z 443.408,A -85,B 0,C 180,E1 12985.294,E2 12985.294} C_VEL
LIN {X 0,Y 298.963,Z 438.661,A -85,B 0,C 180,E1 12983.337,E2 12983.337} C_VEL
LIN {X 0,Y 296.933,Z 436.245,A -85,B 0,C 180,E1 12982.25,E2 12982.25} C_VEL
LIN {X 0,Y 293.663,Z 431.828,A -85,B 0,C 180,E1 12980.311,E2 12980.311} C_VEL
LIN {X 0,Y 290.343,Z 428.139,A -85,B 0,C 180,E1 12978.149,E2 12978.149} C_VEL
LIN {X 0,Y 289.222,Z 426.149,A -85,B 0,C 180,E1 12977.286,E2 12977.286} C_VEL
LIN {X 0,Y 285.91,Z 423.118,A -85,B 0,C 180,E1 12974.677,E2 12974.677} C_VEL
LIN {X 0,Y 284.268,Z 420.091,A -85,B 0,C 180,E1 12972.999,E2 12972.999} C_VEL
LIN {X 0,Y 280.447,Z 417.037,A -85,B 0,C 180,E1 12968.396,E2 12968.396} C_VEL
LIN {X 0,Y 278.909,Z 413.976,A -85,B 0,C 180,E1 12964.926,E2 12964.926} C_VEL
LIN {X 0,Y 278.041,Z 413.363,A -85,B 0,C 180,E1 12960.403,E2 12960.403} C_VEL
LIN {X 0,Y 278.847,Z 413.897,A -85,B 0,C 180,E1 12955.673,E2 12955.673} C_VEL
LIN {X 0,Y 279.575,Z 415.395,A -85,B 0,C 180,E1 12953.729,E2 12953.729} C_VEL
LIN {X 0,Y 282.198,Z 418.914,A -85,B 0,C 180,E1 12949.581,E2 12949.581} C_VEL
LIN {X 0,Y 284.473,Z 420.426,A -85,B 0,C 180,E1 12947.199,E2 12947.199} C_VEL
LIN {X 0,Y 286.709,Z 424.137,A -85,B 0,C 180,E1 12945.037,E2 12945.037} C_VEL
LIN {X 0,Y 289.618,Z 426.797,A -85,B 0,C 180,E1 12942.824,E2 12942.824} C_VEL
LIN {X 0,Y 292.768,Z 431.031,A -85,B 0,C 180,E1 12940.646,E2 12940.646} C_VEL
LIN {X 0,Y 294.371,Z 432.73,A -85,B 0,C 180,E1 12939.67,E2 12939.67} C_VEL
LIN {X 0,Y 297.807,Z 437.169,A -85,B 0,C 180,E1 12937.697,E2 12937.697} C_VEL
LIN {X 0,Y 300.109,Z 440.253,A -85,B 0,C 180,E1 12936.479,E2 12936.479} C_VEL
LIN {X 0,Y 303.282,Z 444.317,A -85,B 0,C 180,E1 12934.928,E2 12934.928} C_VEL
LIN {X 0,Y 308.207,Z 451.045,A -85,B 0,C 180,E1 12932.72,E2 12932.72} C_VEL
LIN {X 0,Y 310.723,Z 454.902,A -85,B 0,C 180,E1 12931.658,E2 12931.658} C_VEL
LIN {X 0,Y 316.214,Z 464.287,A -85,B 0,C 180,E1 12929.469,E2 12929.469} C_VEL
LIN {X 0,Y 318.396,Z 469.874,A -85,B 0,C 180,E1 12928.578,E2 12928.578} C_VEL
LIN {X 0,Y 321.436,Z 483.14,A -85,B 0,C 180,E1 12927.173,E2 12927.173} C_VEL
LIN {X 0,Y 323.779,Z 491.383,A -85,B 0,C 180,E1 12926.219,E2 12926.219} C_VEL
LIN {X 0,Y 324.467,Z 493.018,A -85,B 0,C 180,E1 12925.976,E2 12925.976} C_VEL
LIN {X 0,Y 325.677,Z 495.961,A -85,B 0,C 180,E1 12925.553,E2 12925.553} C_VEL
LIN {X 0,Y 315.945,Z 643.663,A -85,B 0,C 180,E1 12922.364,E2 12922.364} C_VEL
LIN {X 0,Y 313.312,Z 664.954,A -85,B 0,C 180,E1 12921.705,E2 12921.705} C_VEL
LIN {X 0,Y 310.055,Z 682.797,A -85,B 0,C 180,E1 12920.92,E2 12920.92} C_VEL
LIN {X 0,Y 306.308,Z 699.582,A -85,B 0,C 180,E1 12919.96,E2 12919.96} C_VEL
LIN {X 0,Y 301.317,Z 718.532,A -85,B 0,C 180,E1 12918.583,E2 12918.583} C_VEL
LIN {X 0,Y 295.713,Z 736.28,A -85,B 0,C 180,E1 12916.913,E2 12916.913} C_VEL
LIN {X 0,Y 290.651,Z 750.706,A -85,B 0,C 180,E1 12915.264,E2 12915.264} C_VEL
LIN {X 0,Y 284.368,Z 767.158,A -85,B 0,C 180,E1 12912.992,E2 12912.992} C_VEL
LIN {X 0,Y 277.934,Z 782.401,A -85,B 0,C 180,E1 12910.355,E2 12910.355} C_VEL
LIN {X 0,Y 272.493,Z 794.721,A -85,B 0,C 180,E1 12907.789,E2 12907.789} C_VEL
LIN {X 0,Y 266.547,Z 807.869,A -85,B 0,C 180,E1 12904.5,E2 12904.5} C_VEL
LIN {X 0,Y 261.154,Z 819.46,A -85,B 0,C 180,E1 12900.865,E2 12900.865} C_VEL
LIN {X 0,Y 257.217,Z 828.215,A -85,B 0,C 180,E1 12897.553,E2 12897.553} C_VEL
LIN {X 0,Y 253.499,Z 837.109,A -85,B 0,C 180,E1 12893.475,E2 12893.475} C_VEL
LIN {X 0,Y 250.68,Z 844.628,A -85,B 0,C 180,E1 12889.021,E2 12889.021} C_VEL
LIN {X 0,Y 249.13,Z 849.776,A -85,B 0,C 180,E1 12885.121,E2 12885.121} C_VEL
LIN {X 0,Y 248.285,Z 853.776,A -85,B 0,C 180,E1 12881.145,E2 12881.145} C_VEL
LIN {X 0,Y 247.973,Z 856.946,A -85,B 0,C 180,E1 12876.482,E2 12876.482} C_VEL
LIN {X 0,Y 247.98,Z 858.283,A -85,B 0,C 180,E1 12872.311,E2 12872.311} C_VEL
LIN {X 0,Y 247.995,Z 858.433,A -85,B 0,C 180,E1 12868.845,E2 12868.845} C_VEL
LIN {X 0,Y 247.963,Z 857.576,A -85,B 0,C 180,E1 12865.143,E2 12865.143} C_VEL
LIN {X 0,Y 248.048,Z 855.678,A -85,B 0,C 180,E1 12861.423,E2 12861.423} C_VEL
LIN {X 0,Y 248.51,Z 852.512,A -85,B 0,C 180,E1 12857.452,E2 12857.452} C_VEL
LIN {X 0,Y 249.969,Z 846.886,A -85,B 0,C 180,E1 12852.543,E2 12852.543} C_VEL
LIN {X 0,Y 252.037,Z 840.797,A -85,B 0,C 180,E1 12848.595,E2 12848.595} C_VEL
LIN {X 0,Y 254.813,Z 833.81,A -85,B 0,C 180,E1 12844.927,E2 12844.927} C_VEL
LIN {X 0,Y 258.968,Z 824.403,A -85,B 0,C 180,E1 12840.892,E2 12840.892} C_VEL
LIN {X 0,Y 263.883,Z 813.522,A -85,B 0,C 180,E1 12837.193,E2 12837.193} C_VEL
LIN {X 0,Y 268.737,Z 802.969,A -85,B 0,C 180,E1 12834.212,E2 12834.212} C_VEL
LIN {X 0,Y 274.525,Z 790.258,A -85,B 0,C 180,E1 12831.213,E2 12831.213} C_VEL
LIN {X 0,Y 281.089,Z 775.006,A -85,B 0,C 180,E1 12828.306,E2 12828.306} C_VEL
LIN {X 0,Y 286.59,Z 761.405,A -85,B 0,C 180,E1 12826.171,E2 12826.171} C_VEL
LIN {X 0,Y 292.22,Z 746.433,A -85,B 0,C 180,E1 12824.209,E2 12824.209} C_VEL
LIN {X 0,Y 298.473,Z 727.761,A -85,B 0,C 180,E1 12822.242,E2 12822.242} C_VEL
LIN {X 0,Y 303.032,Z 712.186,A -85,B 0,C 180,E1 12820.925,E2 12820.925} C_VEL
LIN {X 0,Y 307.178,Z 695.972,A -85,B 0,C 180,E1 12819.812,E2 12819.812} C_VEL
LIN {X 0,Y 311.55,Z 675.254,A -85,B 0,C 180,E1 12818.718,E2 12818.718} C_VEL
LIN {X 0,Y 314.481,Z 656.596,A -85,B 0,C 180,E1 12818.013,E2 12818.013} C_VEL
LIN {X 0,Y 316.382,Z 638.576,A -85,B 0,C 180,E1 12817.509,E2 12817.509} C_VEL
LIN {X 0,Y 325.608,Z 495.431,A -85,B 0,C 180,E1 12814.41,E2 12814.41} C_VEL
LIN {X 0,Y 318.732,Z 481.296,A -85,B 0,C 180,E1 12811.996,E2 12811.996} C_VEL
LIN {X 0,Y 311.523,Z 467.723,A -85,B 0,C 180,E1 12809.207,E2 12809.207} C_VEL
LIN {X 0,Y 306.022,Z 458.456,A -85,B 0,C 180,E1 12806.86,E2 12806.86} C_VEL
LIN {X 0,Y 299.759,Z 449.672,A -85,B 0,C 180,E1 12803.915,E2 12803.915} C_VEL
LIN {X 0,Y 295.663,Z 444.375,A -85,B 0,C 180,E1 12801.742,E2 12801.742} C_VEL
LIN {X 0,Y 291.662,Z 439.136,A -85,B 0,C 180,E1 12799.326,E2 12799.326} C_VEL
LIN {X 0,Y 288.228,Z 434.845,A -85,B 0,C 180,E1 12796.949,E2 12796.949} C_VEL
LIN {X 0,Y 287.484,Z 433.771,A -85,B 0,C 180,E1 12796.37,E2 12796.37} C_VEL
LIN {X 0,Y 284.11,Z 430.238,A -85,B 0,C 180,E1 12793.543,E2 12793.543} C_VEL
LIN {X 0,Y 282.923,Z 427.844,A -85,B 0,C 180,E1 12792.25,E2 12792.25} C_VEL
LIN {X 0,Y 279.477,Z 425.132,A -85,B 0,C 180,E1 12788.029,E2 12788.029} C_VEL
LIN {X 0,Y 277.94,Z 421.964,A -85,B 0,C 180,E1 12784.548,E2 12784.548} C_VEL
LIN {X 0,Y 277.074,Z 421.291,A -85,B 0,C 180,E1 12780.216,E2 12780.216} C_VEL
LIN {X 0,Y 277.795,Z 421.796,A -85,B 0,C 180,E1 12775.468,E2 12775.468} C_VEL
LIN {X 0,Y 278.578,Z 423.475,A -85,B 0,C 180,E1 12773.311,E2 12773.311} C_VEL
LIN {X 0,Y 281.566,Z 427.121,A -85,B 0,C 180,E1 12768.747,E2 12768.747} C_VEL
LIN {X 0,Y 283.082,Z 428.167,A -85,B 0,C 180,E1 12767.153,E2 12767.153} C_VEL
LIN {X 0,Y 285.602,Z 432.173,A -85,B 0,C 180,E1 12764.684,E2 12764.684} C_VEL
LIN {X 0,Y 287.902,Z 434.29,A -85,B 0,C 180,E1 12762.893,E2 12762.893} C_VEL
LIN {X 0,Y 290.887,Z 438.463,A -85,B 0,C 180,E1 12760.743,E2 12760.743} C_VEL
LIN {X 0,Y 292.604,Z 440.285,A -85,B 0,C 180,E1 12759.664,E2 12759.664} C_VEL
LIN {X 0,Y 297.124,Z 446.324,A -85,B 0,C 180,E1 12757.034,E2 12757.034} C_VEL
LIN {X 0,Y 301.415,Z 451.294,A -85,B 0,C 180,E1 12754.886,E2 12754.886} C_VEL
LIN {X 0,Y 306.486,Z 457.058,A -85,B 0,C 180,E1 12752.625,E2 12752.625} C_VEL
LIN {X 0,Y 310.145,Z 460.258,A -85,B 0,C 180,E1 12751.145,E2 12751.145} C_VEL
LIN {X 0,Y 315.391,Z 465.16,A -85,B 0,C 180,E1 12748.898,E2 12748.898} C_VEL
LIN {X 0,Y 318.972,Z 467.988,A -85,B 0,C 180,E1 12747.279,E2 12747.279} C_VEL
LIN {X 0,Y 323.48,Z 472.352,A -85,B 0,C 180,E1 12745.027,E2 12745.027} C_VEL
LIN {X 0,Y 326.809,Z 474.977,A -85,B 0,C 180,E1 12743.279,E2 12743.279} C_VEL
LIN {X 0,Y 330.733,Z 479.234,A -85,B 0,C 180,E1 12740.939,E2 12740.939} C_VEL
LIN {X 0,Y 334.34,Z 482.309,A -85,B 0,C 180,E1 12738.758,E2 12738.758} C_VEL
LIN {X 0,Y 338.601,Z 486.876,A -85,B 0,C 180,E1 12736.072,E2 12736.072} C_VEL
LIN {X 0,Y 341.725,Z 489.345,A -85,B 0,C 180,E1 12734.1,E2 12734.1} C_VEL
LIN {X 0,Y 345.577,Z 493.612,A -85,B 0,C 180,E1 12731.48,E2 12731.48} C_VEL
LIN {X 0,Y 349.475,Z 496.648,A -85,B 0,C 180,E1 12728.845,E2 12728.845} C_VEL
LIN {X 0,Y 353.32,Z 500.902,A -85,B 0,C 180,E1 12725.985,E2 12725.985} C_VEL
LIN {X 0,Y 357.487,Z 503.985,A -85,B 0,C 180,E1 12722.82,E2 12722.82} C_VEL
LIN {X 0,Y 360.647,Z 507.696,A -85,B 0,C 180,E1 12720.118,E2 12720.118} C_VEL
LIN {X 0,Y 364.051,Z 510.282,A -85,B 0,C 180,E1 12717.123,E2 12717.123} C_VEL
LIN {X 0,Y 365.88,Z 511.459,A -85,B 0,C 180,E1 12715.406,E2 12715.406} C_VEL
LIN {X 0,Y 368.381,Z 514.721,A -85,B 0,C 180,E1 12712.669,E2 12712.669} C_VEL
LIN {X 0,Y 371.12,Z 517.056,A -85,B 0,C 180,E1 12709.478,E2 12709.478} C_VEL
LIN {X 0,Y 373.658,Z 518.341,A -85,B 0,C 180,E1 12706.158,E2 12706.158} C_VEL
LIN {X 0,Y 374.893,Z 519.307,A -85,B 0,C 180,E1 12704.203,E2 12704.203} C_VEL
LIN {X 0,Y 376.424,Z 521.721,A -85,B 0,C 180,E1 12701.025,E2 12701.025} C_VEL
LIN {X 0,Y 377.667,Z 523.113,A -85,B 0,C 180,E1 12697.76,E2 12697.76} C_VEL
LIN {X 0,Y 378.545,Z 523.88,A -85,B 0,C 180,E1 12694.393,E2 12694.393} C_VEL
LIN {X 0,Y 378.903,Z 524.14,A -85,B 0,C 180,E1 12691.058,E2 12691.058} C_VEL
LIN {X 0,Y 378.83,Z 524.119,A -85,B 0,C 180,E1 12687.731,E2 12687.731} C_VEL
LIN {X 0,Y 378.261,Z 523.654,A -85,B 0,C 180,E1 12684.388,E2 12684.388} C_VEL
LIN {X 0,Y 377.176,Z 522.657,A -85,B 0,C 180,E1 12680.848,E2 12680.848} C_VEL
LIN {X 0,Y 375.768,Z 520.765,A -85,B 0,C 180,E1 12677.512,E2 12677.512} C_VEL
LIN {X 0,Y 374.283,Z 518.63,A -85,B 0,C 180,E1 12674.824,E2 12674.824} C_VEL
LIN {X 0,Y 371.899,Z 517.517,A -85,B 0,C 180,E1 12671.504,E2 12671.504} C_VEL
LIN {X 0,Y 369.186,Z 515.519,A -85,B 0,C 180,E1 12668.241,E2 12668.241} C_VEL
LIN {X 0,Y 366.487,Z 512.422,A -85,B 0,C 180,E1 12665.273,E2 12665.273} C_VEL
LIN {X 0,Y 365.304,Z 510.922,A -85,B 0,C 180,E1 12664.029,E2 12664.029} C_VEL
LIN {X 0,Y 362.041,Z 508.916,A -85,B 0,C 180,E1 12661.079,E2 12661.079} C_VEL
LIN {X 0,Y 358.697,Z 505.607,A -85,B 0,C 180,E1 12658.209,E2 12658.209} C_VEL
LIN {X 0,Y 356.778,Z 503.316,A -85,B 0,C 180,E1 12656.611,E2 12656.611} C_VEL
LIN {X 0,Y 353.029,Z 500.639,A -85,B 0,C 180,E1 12653.804,E2 12653.804} C_VEL
LIN {X 0,Y 349.123,Z 496.168,A -85,B 0,C 180,E1 12650.89,E2 12650.89} C_VEL
LIN {X 0,Y 344.861,Z 492.946,A -85,B 0,C 180,E1 12648.03,E2 12648.03} C_VEL
LIN {X 0,Y 340.994,Z 488.594,A -85,B 0,C 180,E1 12645.426,E2 12645.426} C_VEL
LIN {X 0,Y 336.963,Z 485.339,A -85,B 0,C 180,E1 12642.907,E2 12642.907} C_VEL
LIN {X 0,Y 333.172,Z 481.152,A -85,B 0,C 180,E1 12640.507,E2 12640.507} C_VEL
LIN {X 0,Y 328.467,Z 477.008,A -85,B 0,C 180,E1 12637.71,E2 12637.71} C_VEL
LIN {X 0,Y 325.686,Z 473.962,A -85,B 0,C 180,E1 12636.105,E2 12636.105} C_VEL
LIN {X 0,Y 320.902,Z 470.038,A -85,B 0,C 180,E1 12633.672,E2 12633.672} C_VEL
LIN {X 0,Y 317.506,Z 466.658,A -85,B 0,C 180,E1 12632.036,E2 12632.036} C_VEL
LIN {X 0,Y 312.424,Z 462.622,A -85,B 0,C 180,E1 12629.833,E2 12629.833} C_VEL
LIN {X 0,Y 307.969,Z 458.257,A -85,B 0,C 180,E1 12627.967,E2 12627.967} C_VEL
LIN {X 0,Y 302.807,Z 453.16,A -85,B 0,C 180,E1 12625.776,E2 12625.776} C_VEL
LIN {X 0,Y 300.282,Z 450.238,A -85,B 0,C 180,E1 12624.585,E2 12624.585} C_VEL
LIN {X 0,Y 295.473,Z 444.151,A -85,B 0,C 180,E1 12622.052,E2 12622.052} C_VEL
LIN {X 0,Y 291.786,Z 439.274,A -85,B 0,C 180,E1 12619.82,E2 12619.82} C_VEL
LIN {X 0,Y 288.447,Z 435.293,A -85,B 0,C 180,E1 12617.542,E2 12617.542} C_VEL
LIN {X 0,Y 287.468,Z 433.696,A -85,B 0,C 180,E1 12616.769,E2 12616.769} C_VEL
LIN {X 0,Y 284.296,Z 430.507,A -85,B 0,C 180,E1 12614.138,E2 12614.138} C_VEL
LIN {X 0,Y 282.898,Z 427.889,A -85,B 0,C 180,E1 12612.648,E2 12612.648} C_VEL
LIN {X 0,Y 279.231,Z 424.752,A -85,B 0,C 180,E1 12608.018,E2 12608.018} C_VEL
LIN {X 0,Y 277.864,Z 421.865,A -85,B 0,C 180,E1 12604.738,E2 12604.738} C_VEL
LIN {X 0,Y 277.074,Z 421.291,A -85,B 0,C 180,E1 12599.784,E2 12599.784} C_VEL
LIN {X 0,Y 277.94,Z 421.963,A -85,B 0,C 180,E1 12595.452,E2 12595.452} C_VEL
